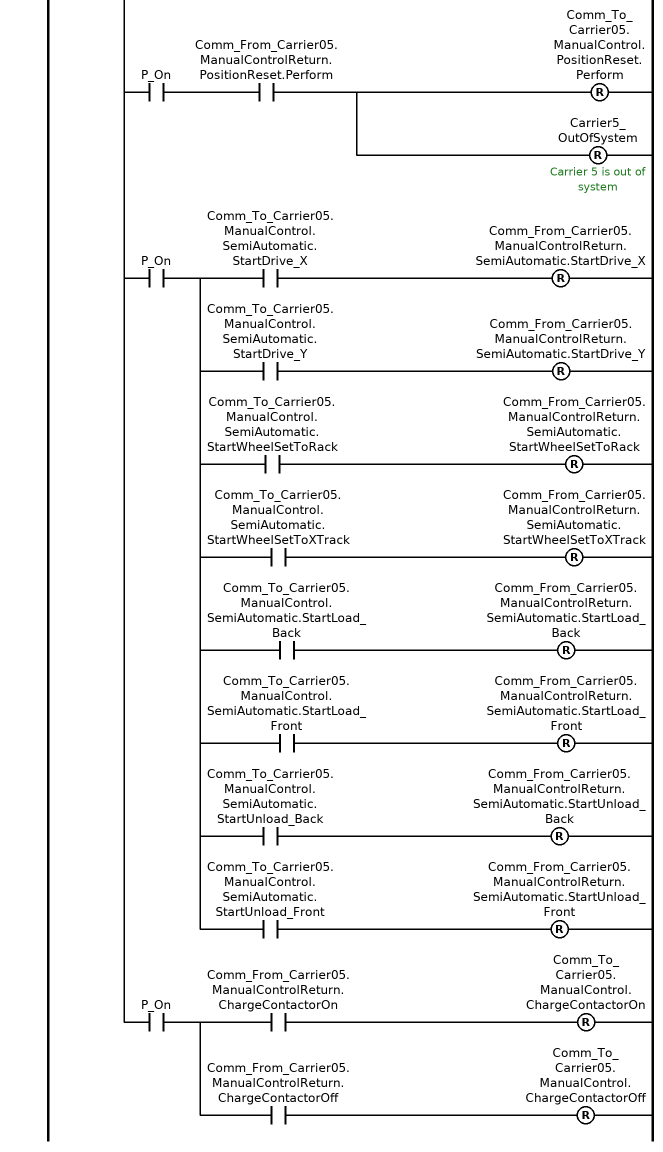
(* [picture p78: Mobile_Machines / Carrier05, rungs 8-8] *)
(* Rung 8: Reset several bits that are set by Dat-A-Control but not reset *)
IF P_On AND P_On AND Comm_From_Carrier05.Various.ResetAlarm_Return THEN
    Comm_To_Carrier05.Dat_A_Control.Settings_In0.ResetAlarm := FALSE;
END_IF;
IF P_On AND P_On AND Comm_From_Carrier05.Various.ResetCycle_Return THEN
    Comm_To_Carrier05.Dat_A_Control.Settings_In0.ResetCycle := FALSE;
END_IF;
IF P_On AND P_On AND Comm_From_Carrier05.Various.AbortCharge_Return THEN
    Comm_To_Carrier05.Various.AbortCharge := FALSE;
END_IF;
IF P_On AND P_On AND ES_OK AND Comm_From_Carrier05.Various.ResetMachineOn THEN
    Comm_To_Carrier05.Dat_A_Control.Settings_In0.MachineOn := FALSE;
END_IF;
IF P_On AND P_On AND Comm_From_Carrier05.ManualControlReturn.DriveRack.Out THEN
    Comm_To_Carrier05.ManualControl.DriveRack.Out := FALSE;
END_IF;
IF P_On AND P_On AND Comm_From_Carrier05.ManualControlReturn.DriveRack.In THEN
    Comm_To_Carrier05.ManualControl.DriveRack.In := FALSE;
END_IF;
IF P_On AND P_On AND Comm_From_Carrier05.ManualControlReturn.DriveRack.Stop THEN
    Comm_To_Carrier05.ManualControl.DriveRack.Stop := FALSE;
END_IF;
IF P_On AND P_On AND Comm_From_Carrier05.ManualControlReturn.DriveRack_FindXTrack.Out THEN
    Comm_To_Carrier05.ManualControl.DriveRack_FindXTrack.Out := FALSE;
END_IF;
IF P_On AND P_On AND Comm_From_Carrier05.ManualControlReturn.DriveRack_FindXTrack.In THEN
    Comm_To_Carrier05.ManualControl.DriveRack_FindXTrack.In := FALSE;
END_IF;
IF P_On AND P_On AND Comm_From_Carrier05.ManualControlReturn.DriveRack_FindXTrack.Stop THEN
    Comm_To_Carrier05.ManualControl.DriveRack_FindXTrack.Stop := FALSE;
END_IF;
IF P_On AND P_On AND Comm_From_Carrier05.ManualControlReturn.DriveXtrack.Out THEN
    Comm_To_Carrier05.ManualControl.DriveXtrack.Out := FALSE;
END_IF;
IF P_On AND P_On AND Comm_From_Carrier05.ManualControlReturn.DriveXtrack.In THEN
    Comm_To_Carrier05.ManualControl.DriveXtrack.In := FALSE;
END_IF;
IF P_On AND P_On AND Comm_From_Carrier05.ManualControlReturn.DriveXtrack.Stop THEN
    Comm_To_Carrier05.ManualControl.DriveXtrack.Stop := FALSE;
END_IF;
IF P_On AND P_On AND Comm_From_Carrier05.ManualControlReturn.DriveXTrack_FindPosition.Out THEN
    Comm_To_Carrier05.ManualControl.DriveXTrack_FindPosition.Out := FALSE;
END_IF;
IF P_On AND P_On AND Comm_From_Carrier05.ManualControlReturn.DriveXTrack_FindPosition.In THEN
    Comm_To_Carrier05.ManualControl.DriveXTrack_FindPosition.In := FALSE;
END_IF;
IF P_On AND P_On AND Comm_From_Carrier05.ManualControlReturn.DriveXTrack_FindPosition.Stop THEN
    Comm_To_Carrier05.ManualControl.DriveXTrack_FindPosition.Stop := FALSE;
END_IF;
IF P_On AND P_On AND Comm_From_Carrier05.ManualControlReturn.Wheelset.Out THEN
    Comm_To_Carrier05.ManualControl.Wheelset.Out := FALSE;
END_IF;
IF P_On AND P_On AND Comm_From_Carrier05.ManualControlReturn.Wheelset.In THEN
    Comm_To_Carrier05.ManualControl.Wheelset.In := FALSE;
END_IF;
IF P_On AND P_On AND Comm_From_Carrier05.ManualControlReturn.Wheelset.Stop THEN
    Comm_To_Carrier05.ManualControl.Wheelset.Stop := FALSE;
END_IF;
IF P_On AND P_On AND Comm_From_Carrier05.ManualControlReturn.LIftingPlate.UpMIN THEN
    Comm_To_Carrier05.ManualControl.LIftingPlate.UpMIN := FALSE;
END_IF;
IF P_On AND P_On AND Comm_From_Carrier05.ManualControlReturn.LIftingPlate.DownMIN THEN
    Comm_To_Carrier05.ManualControl.LIftingPlate.DownMIN := FALSE;
END_IF;
IF P_On AND P_On AND Comm_From_Carrier05.ManualControlReturn.LIftingPlate.StopMIN THEN
    Comm_To_Carrier05.ManualControl.LIftingPlate.StopMIN := FALSE;
END_IF;
IF P_On AND P_On AND Comm_From_Carrier05.ManualControlReturn.LIftingPlate.UpMAX THEN
    Comm_To_Carrier05.ManualControl.LIftingPlate.UpMAX := FALSE;
END_IF;
IF P_On AND P_On AND Comm_From_Carrier05.ManualControlReturn.LIftingPlate.DownMAX THEN
    Comm_To_Carrier05.ManualControl.LIftingPlate.DownMAX := FALSE;
END_IF;
IF P_On AND P_On AND Comm_From_Carrier05.ManualControlReturn.LIftingPlate.StopMAX THEN
    Comm_To_Carrier05.ManualControl.LIftingPlate.StopMAX := FALSE;
END_IF;
IF P_On AND P_On AND Comm_From_Carrier05.ManualControlReturn.LIftingPlate.UpBoth THEN
    Comm_To_Carrier05.ManualControl.LIftingPlate.UpBoth := FALSE;
END_IF;
IF P_On AND P_On AND Comm_From_Carrier05.ManualControlReturn.LIftingPlate.DownBoth THEN
    Comm_To_Carrier05.ManualControl.LIftingPlate.DownBoth := FALSE;
END_IF;
IF P_On AND P_On AND Comm_From_Carrier05.ManualControlReturn.LIftingPlate.StopBoth THEN
    Comm_To_Carrier05.ManualControl.LIftingPlate.StopBoth := FALSE;
END_IF;
_p59 := P_On AND P_On AND Comm_From_Carrier05.ManualControlReturn.PositionReset.Perform;
IF _p59 THEN
    Comm_To_Carrier05.ManualControl.PositionReset.Perform := FALSE;
    Carrier5_OutOfSystem := FALSE;
END_IF;
IF P_On AND P_On AND Comm_To_Carrier05.ManualControl.SemiAutomatic.StartDrive_X THEN
    Comm_From_Carrier05.ManualControlReturn.SemiAutomatic.StartDrive_X := FALSE;
END_IF;
IF P_On AND P_On AND Comm_To_Carrier05.ManualControl.SemiAutomatic.StartDrive_Y THEN
    Comm_From_Carrier05.ManualControlReturn.SemiAutomatic.StartDrive_Y := FALSE;
END_IF;
IF P_On AND P_On AND Comm_To_Carrier05.ManualControl.SemiAutomatic.StartWheelSetToRack THEN
    Comm_From_Carrier05.ManualControlReturn.SemiAutomatic.StartWheelSetToRack := FALSE;
END_IF;
IF P_On AND P_On AND Comm_To_Carrier05.ManualControl.SemiAutomatic.StartWheelSetToXTrack THEN
    Comm_From_Carrier05.ManualControlReturn.SemiAutomatic.StartWheelSetToXTrack := FALSE;
END_IF;
IF P_On AND P_On AND Comm_To_Carrier05.ManualControl.SemiAutomatic.StartLoad_Back THEN
    Comm_From_Carrier05.ManualControlReturn.SemiAutomatic.StartLoad_Back := FALSE;
END_IF;
IF P_On AND P_On AND Comm_To_Carrier05.ManualControl.SemiAutomatic.StartLoad_Front THEN
    Comm_From_Carrier05.ManualControlReturn.SemiAutomatic.StartLoad_Front := FALSE;
END_IF;
IF P_On AND P_On AND Comm_To_Carrier05.ManualControl.SemiAutomatic.StartUnload_Back THEN
    Comm_From_Carrier05.ManualControlReturn.SemiAutomatic.StartUnload_Back := FALSE;
END_IF;
IF P_On AND P_On AND Comm_To_Carrier05.ManualControl.SemiAutomatic.StartUnload_Front THEN
    Comm_From_Carrier05.ManualControlReturn.SemiAutomatic.StartUnload_Front := FALSE;
END_IF;
IF P_On AND P_On AND Comm_From_Carrier05.ManualControlReturn.ChargeContactorOn THEN
    Comm_To_Carrier05.ManualControl.ChargeContactorOn := FALSE;
END_IF;
IF P_On AND P_On AND Comm_From_Carrier05.ManualControlReturn.ChargeContactorOff THEN
    Comm_To_Carrier05.ManualControl.ChargeContactorOff := FALSE;
END_IF;

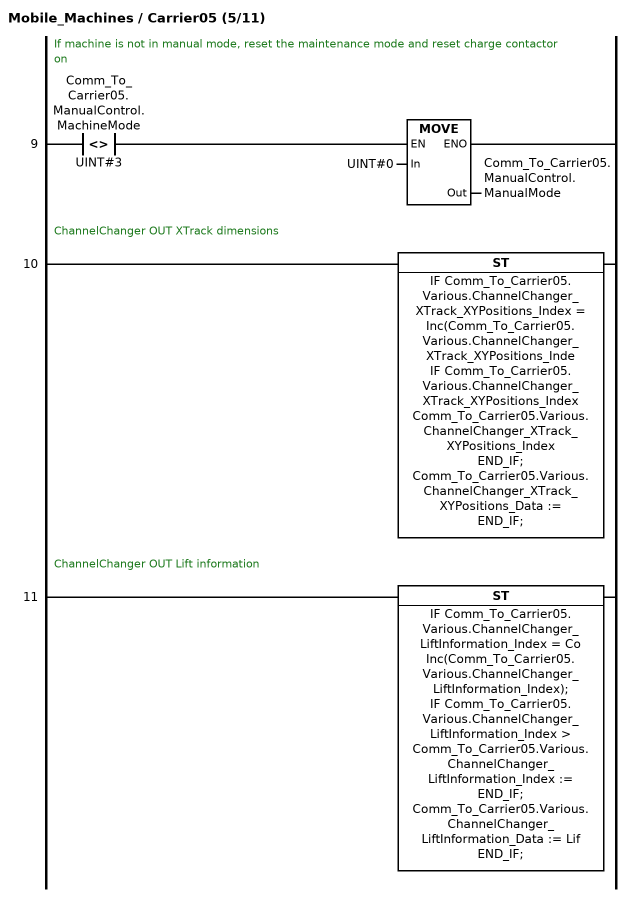
(* Rung 9: If machine is not in manual mode, reset the maintenance mode and reset charge contactor on *)
IF Comm_To_Carrier05.ManualControl.MachineMode <> UINT#3 THEN
    Comm_To_Carrier05.ManualControl.ManualMode := UINT#0;
END_IF;
(* Rung 10: ChannelChanger OUT XTrack dimensions *)
IF Comm_To_Carrier05.Various.ChannelChanger_XTrack_XYPositions_Index = Comm_From_Carrier05.Various.ChannelChanger_XTrack_XYPositions_Index THEN
	Inc(Comm_To_Carrier05.Various.ChannelChanger_XTrack_XYPositions_Index);
	IF Comm_To_Carrier05.Various.ChannelChanger_XTrack_XYPositions_Index > 199 THEN
		Comm_To_Carrier05.Various.ChannelChanger_XTrack_XYPositions_Index := 0;
	END_IF;
	Comm_To_Carrier05.Various.ChannelChanger_XTrack_XYPositions_Data := XTrack_XYPositions_Array[Comm_To_Carrier05.Various.ChannelChanger_XTrack_XYPositions_Index];
END_IF;
(* Rung 11: ChannelChanger OUT Lift information *)
IF Comm_To_Carrier05.Various.ChannelChanger_LiftInformation_Index = Comm_From_Carrier05.Various.ChannelChanger_LiftInformation_Index THEN
	Inc(Comm_To_Carrier05.Various.ChannelChanger_LiftInformation_Index);
	IF Comm_To_Carrier05.Various.ChannelChanger_LiftInformation_Index > 99 THEN
		Comm_To_Carrier05.Various.ChannelChanger_LiftInformation_Index := 0;
	END_IF;
	Comm_To_Carrier05.Various.ChannelChanger_LiftInformation_Data := Lift_Array[Comm_To_Carrier05.Various.ChannelChanger_LiftInformation_Index];
END_IF;

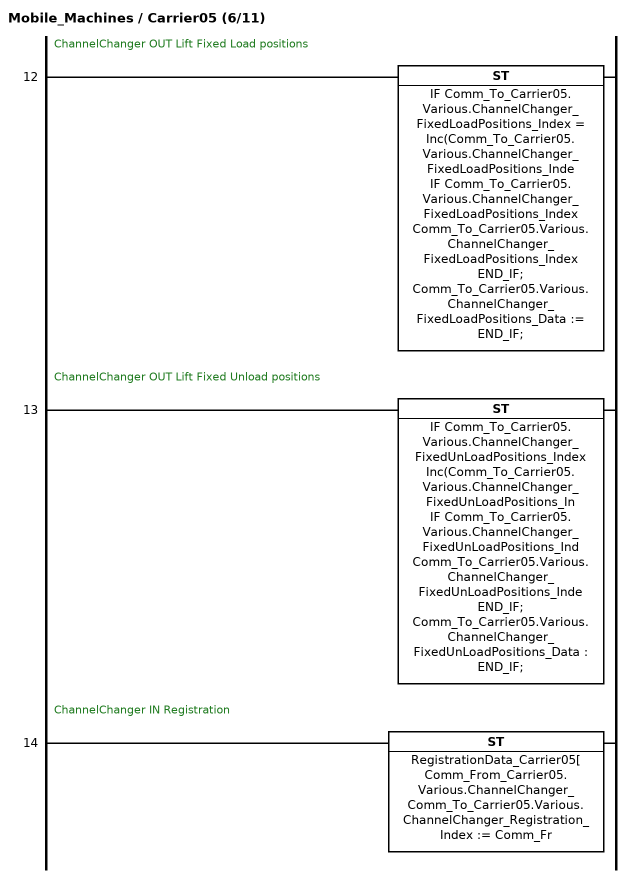
(* Rung 12: ChannelChanger OUT Lift Fixed Load positions *)
IF Comm_To_Carrier05.Various.ChannelChanger_FixedLoadPositions_Index = Comm_From_Carrier05.Various.ChannelChanger_FixedLoadPositions_Index THEN
	Inc(Comm_To_Carrier05.Various.ChannelChanger_FixedLoadPositions_Index);
	IF Comm_To_Carrier05.Various.ChannelChanger_FixedLoadPositions_Index > 199 THEN
		Comm_To_Carrier05.Various.ChannelChanger_FixedLoadPositions_Index := 0;
	END_IF;
	Comm_To_Carrier05.Various.ChannelChanger_FixedLoadPositions_Data := FixedLoadPosition_Array[Comm_To_Carrier05.Various.ChannelChanger_FixedLoadPositions_Index];
END_IF;
(* Rung 13: ChannelChanger OUT Lift Fixed Unload positions *)
IF Comm_To_Carrier05.Various.ChannelChanger_FixedUnLoadPositions_Index = Comm_From_Carrier05.Various.ChannelChanger_FixedUnLoadPositions_Index THEN
	Inc(Comm_To_Carrier05.Various.ChannelChanger_FixedUnLoadPositions_Index);
	IF Comm_To_Carrier05.Various.ChannelChanger_FixedUnLoadPositions_Index > 199 THEN
		Comm_To_Carrier05.Various.ChannelChanger_FixedUnLoadPositions_Index := 0;
	END_IF;
	Comm_To_Carrier05.Various.ChannelChanger_FixedUnLoadPositions_Data := FixedUnloadPosition_Array[Comm_To_Carrier05.Various.ChannelChanger_FixedUnLoadPositions_Index];
END_IF;
(* Rung 14: ChannelChanger IN Registration *)
RegistrationData_Carrier05[Comm_From_Carrier05.Various.ChannelChanger_Registration_Index] := Comm_From_Carrier05.Various.ChannelChanger_Registration_Data;
Comm_To_Carrier05.Various.ChannelChanger_Registration_Index := Comm_From_Carrier05.Various.ChannelChanger_Registration_Index;

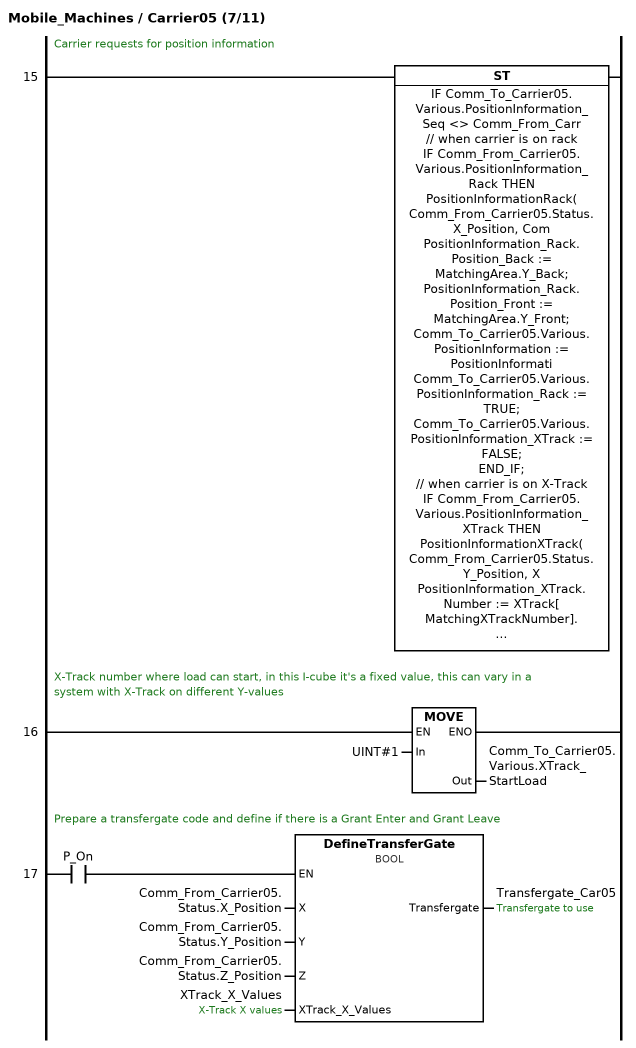
(* Rung 15: Carrier requests for position information *)
IF Comm_To_Carrier05.Various.PositionInformation_Seq <> Comm_From_Carrier05.Various.PositionInformation_Seq THEN
	// when carrier is on rack
	IF Comm_From_Carrier05.Various.PositionInformation_Rack THEN
		PositionInformationRack(Comm_From_Carrier05.Status.X_Position, Comm_From_Carrier05.Status.Y_Position, Comm_From_Carrier05.Status.Z_Position, Settings_CP.Margin_AreaCompare, Area, MatchingArea);
		PositionInformation_Rack.Position_Back := MatchingArea.Y_Back;
		PositionInformation_Rack.Position_Front := MatchingArea.Y_Front;
		Comm_To_Carrier05.Various.PositionInformation := PositionInformation_Rough;
		Comm_To_Carrier05.Various.PositionInformation_Rack := TRUE;
		Comm_To_Carrier05.Various.PositionInformation_XTrack := FALSE;
	END_IF;
	
	// when carrier is on X-Track
	IF Comm_From_Carrier05.Various.PositionInformation_XTrack THEN
		PositionInformationXTrack(Comm_From_Carrier05.Status.Y_Position, XTrack_Y_Values, MatchingXTrackNumber);
		PositionInformation_XTrack.Number := XTrack[MatchingXTrackNumber].XTrack_Number;
		PositionInformation_XTrack.Position_MIN := XTrack[MatchingXTrackNumber].MinimumPosition;
		PositionInformation_XTrack.Position_MAX := XTrack[MatchingXTrackNumber].MaximumPosition;
		Comm_To_Carrier05.Various.PositionInformation := PositionInformation_Rough;
		Comm_To_Carrier05.Various.PositionInformation_Rack := FALSE;
		Comm_To_Carrier05.Various.PositionInformation_XTrack := TRUE;
	END_IF;
	
	Comm_To_Carrier05.Various.PositionInformation_Seq := Comm_From_Carrier05.Various.PositionInformation_Seq;
	
END_IF;
(* Rung 16: X-Track number where load can start, in this I-cube it's a fixed value, this can vary in a system with X-Track on different Y-values *)
Comm_To_Carrier05.Various.XTrack_StartLoad := UINT#1;
(* Rung 17: Prepare a transfergate code and define if there is a Grant Enter and Grant Leave *)
_t60 := FALSE;
IF P_On THEN _t60 := DefineTransferGate(X := Comm_From_Carrier05.Status.X_Position, Y := Comm_From_Carrier05.Status.Y_Position, Z := Comm_From_Carrier05.Status.Z_Position, XTrack_X_Values := XTrack_X_Values, Transfergate => Transfergate_Car05); END_IF;

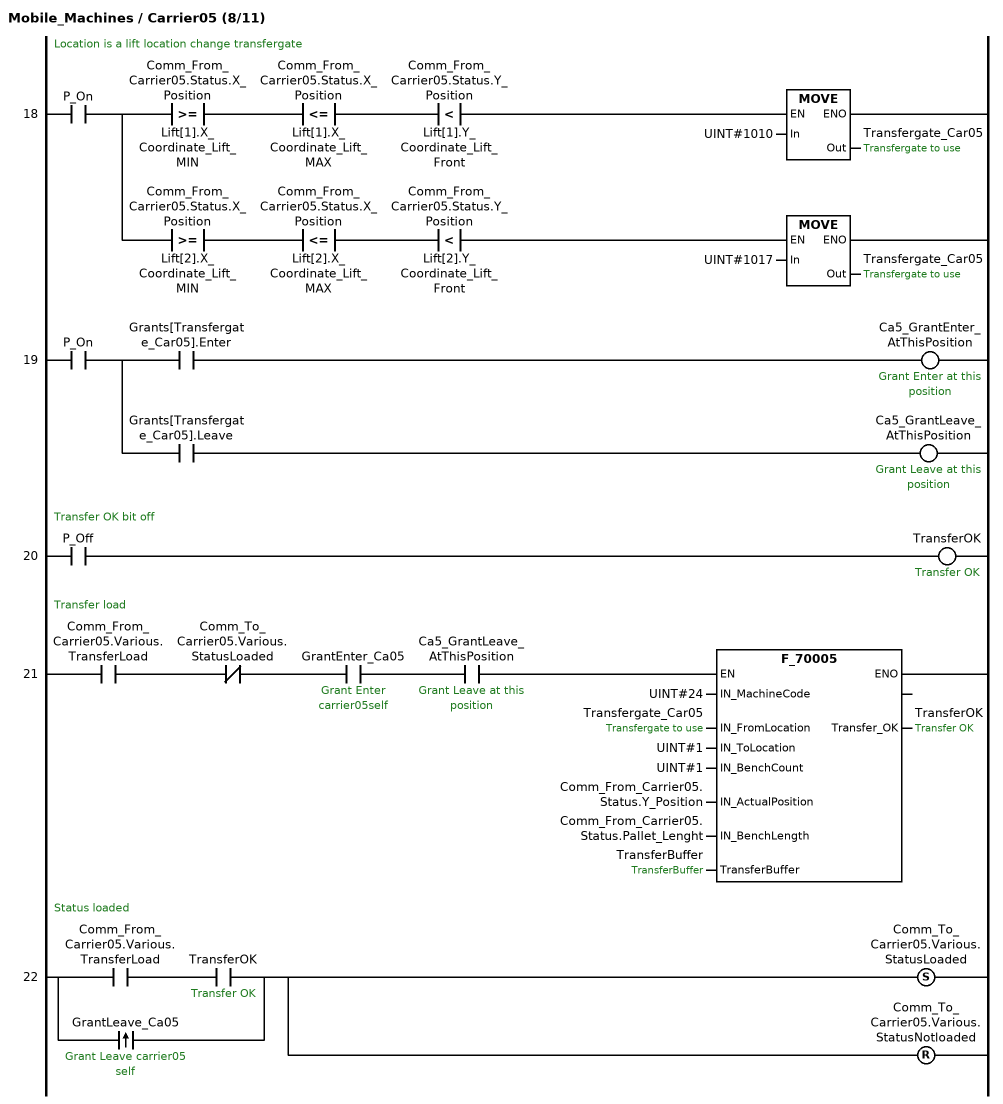
(* Rung 18: Location is a lift location change transfergate *)
IF P_On AND (Comm_From_Carrier05.Status.X_Position >= Lift[1].X_Coordinate_Lift_MIN) AND (Comm_From_Carrier05.Status.X_Position <= Lift[1].X_Coordinate_Lift_MAX) AND (Comm_From_Carrier05.Status.Y_Position < Lift[1].Y_Coordinate_Lift_Front) THEN
    Transfergate_Car05 := UINT#1010;
END_IF;
IF P_On AND (Comm_From_Carrier05.Status.X_Position >= Lift[2].X_Coordinate_Lift_MIN) AND (Comm_From_Carrier05.Status.X_Position <= Lift[2].X_Coordinate_Lift_MAX) AND (Comm_From_Carrier05.Status.Y_Position < Lift[2].Y_Coordinate_Lift_Front) THEN
    Transfergate_Car05 := UINT#1017;
END_IF;
(* Rung 19 *)
Ca5_GrantEnter_AtThisPosition := P_On AND Grants[Transfergate_Car05].Enter;
Ca5_GrantLeave_AtThisPosition := P_On AND Grants[Transfergate_Car05].Leave;
(* Rung 20: Transfer OK bit off *)
TransferOK := P_Off;
(* Rung 21: Transfer load *)
IF Comm_From_Carrier05.Various.TransferLoad AND NOT Comm_To_Carrier05.Various.StatusLoaded AND GrantEnter_Ca05 AND Ca5_GrantLeave_AtThisPosition THEN
    F_70005(IN_MachineCode := UINT#24, IN_FromLocation := Transfergate_Car05, IN_ToLocation := UINT#1, IN_BenchCount := UINT#1, IN_ActualPosition := Comm_From_Carrier05.Status.Y_Position, IN_BenchLength := Comm_From_Carrier05.Status.Pallet_Lenght, TransferBuffer := TransferBuffer, Transfer_OK => TransferOK);
END_IF;
(* Rung 22: Status loaded *)
_e61(CLK := GrantLeave_Ca05);
_p62 := (Comm_From_Carrier05.Various.TransferLoad AND TransferOK) OR _e61.Q;
IF _p62 THEN
    Comm_To_Carrier05.Various.StatusLoaded := TRUE;
    Comm_To_Carrier05.Various.StatusNotloaded := FALSE;
END_IF;

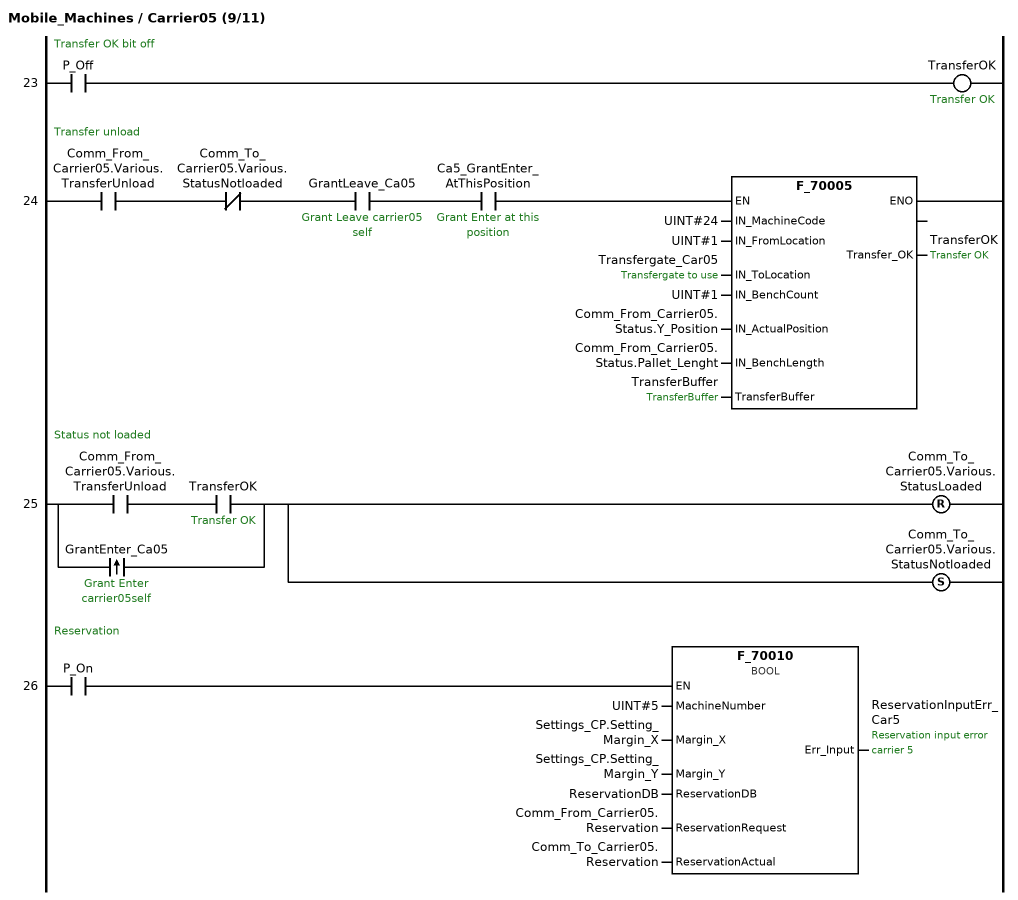
(* Rung 23: Transfer OK bit off *)
TransferOK := P_Off;
(* Rung 24: Transfer unload *)
IF Comm_From_Carrier05.Various.TransferUnload AND NOT Comm_To_Carrier05.Various.StatusNotloaded AND GrantLeave_Ca05 AND Ca5_GrantEnter_AtThisPosition THEN
    F_70005(IN_MachineCode := UINT#24, IN_FromLocation := UINT#1, IN_ToLocation := Transfergate_Car05, IN_BenchCount := UINT#1, IN_ActualPosition := Comm_From_Carrier05.Status.Y_Position, IN_BenchLength := Comm_From_Carrier05.Status.Pallet_Lenght, TransferBuffer := TransferBuffer, Transfer_OK => TransferOK);
END_IF;
(* Rung 25: Status not loaded *)
_e63(CLK := GrantEnter_Ca05);
_p64 := (Comm_From_Carrier05.Various.TransferUnload AND TransferOK) OR _e63.Q;
IF _p64 THEN
    Comm_To_Carrier05.Various.StatusLoaded := FALSE;
    Comm_To_Carrier05.Various.StatusNotloaded := TRUE;
END_IF;
(* Rung 26: Reservation *)
_t65 := FALSE;
IF P_On THEN _t65 := F_70010(MachineNumber := UINT#5, Margin_X := Settings_CP.Setting_Margin_X, Margin_Y := Settings_CP.Setting_Margin_Y, ReservationDB := ReservationDB, ReservationRequest := Comm_From_Carrier05.Reservation, ReservationActual := Comm_To_Carrier05.Reservation, Err_Input => ReservationInputErr_Car5); END_IF;

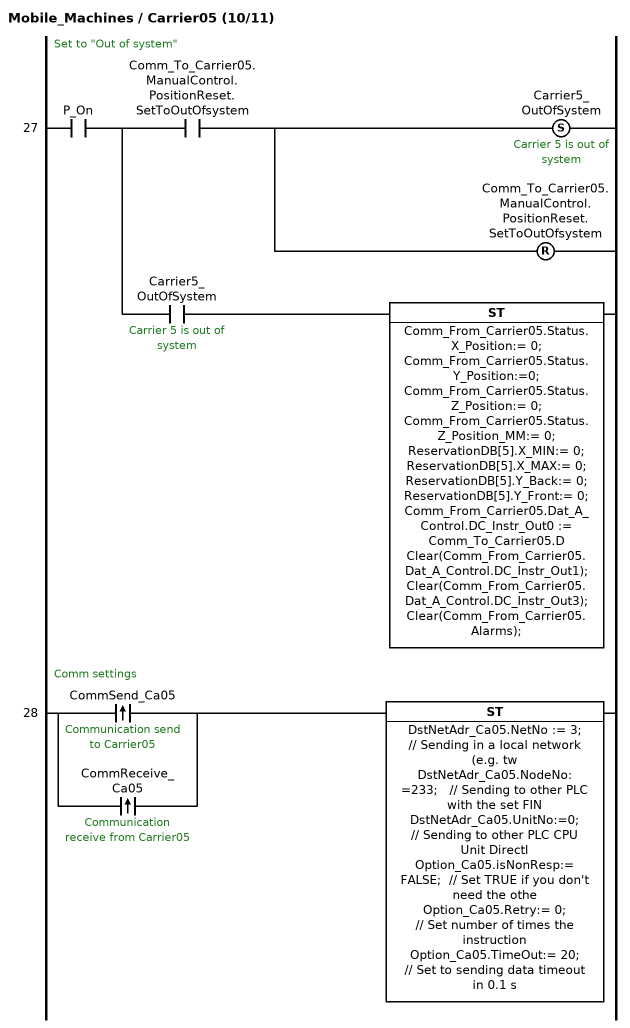
(* Rung 27: Set to "Out of system" *)
_p66 := P_On AND Comm_To_Carrier05.ManualControl.PositionReset.SetToOutOfsystem;
IF _p66 THEN
    Carrier5_OutOfSystem := TRUE;
    Comm_To_Carrier05.ManualControl.PositionReset.SetToOutOfsystem := FALSE;
END_IF;
IF P_On AND Carrier5_OutOfSystem THEN
    Comm_From_Carrier05.Status.X_Position:= 0;
    Comm_From_Carrier05.Status.Y_Position:=0;
    Comm_From_Carrier05.Status.Z_Position:= 0;
    Comm_From_Carrier05.Status.Z_Position_MM:= 0;
    
    ReservationDB[5].X_MIN:= 0;
    ReservationDB[5].X_MAX:= 0;
    ReservationDB[5].Y_Back:= 0;
    ReservationDB[5].Y_Front:= 0;
    
    Comm_From_Carrier05.Dat_A_Control.DC_Instr_Out0 := Comm_To_Carrier05.Dat_A_Control.Instr_Sequencenumber;
    Clear(Comm_From_Carrier05.Dat_A_Control.DC_Instr_Out1);
    Clear(Comm_From_Carrier05.Dat_A_Control.DC_Instr_Out3);
    Clear(Comm_From_Carrier05.Alarms);
END_IF;
(* Rung 28: Comm settings *)
_e67(CLK := CommSend_Ca05);
_e68(CLK := CommReceive_Ca05);
IF _e67.Q OR _e68.Q THEN
    DstNetAdr_Ca05.NetNo := 3;			// Sending in a local network (e.g. two PLCs connected by Ethernet LAN vai a hub)
    DstNetAdr_Ca05.NodeNo:=233;		// Sending to other PLC with the set FINS Node NUmber (depending on the other PLC)
    DstNetAdr_Ca05.UnitNo:=0;			// Sending to other PLC CPU Unit Directly
    
    Option_Ca05.isNonResp:= FALSE; 	// Set TRUE if you don't need the other CPU to reply back, otherwise set to FALSE
    Option_Ca05.Retry:= 0;					// Set number of times the instruction will retry sending if it failed to send data
    Option_Ca05.TimeOut:= 20;			// Set to sending data timeout in 0.1 s unit (e.g. 20 = 2 secs)
END_IF;

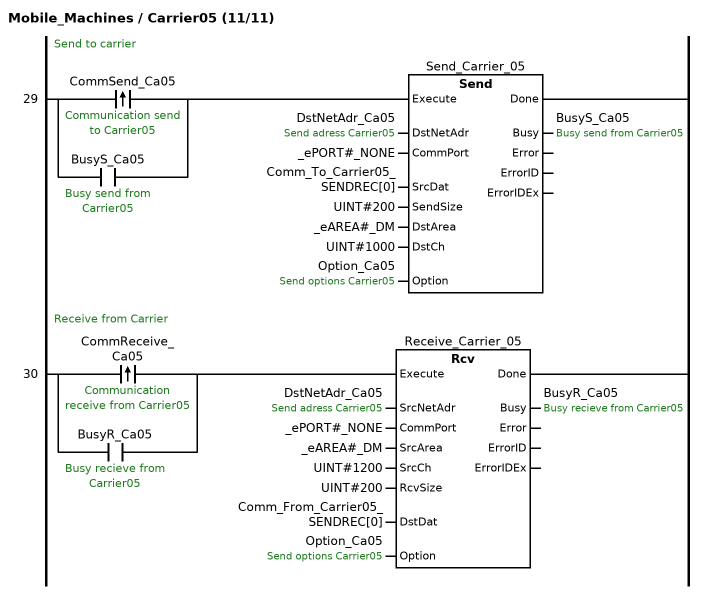
(* Rung 29: Send to carrier *)
_e69(CLK := CommSend_Ca05);
Send_Carrier_05(Execute := _e69.Q OR BusyS_Ca05, DstNetAdr := DstNetAdr_Ca05, CommPort := _ePORT#_NONE, SrcDat := Comm_To_Carrier05_SENDREC[0], SendSize := UINT#200, DstArea := _eAREA#_DM, DstCh := UINT#1000, Option := Option_Ca05, Busy => BusyS_Ca05);
(* Rung 30: Receive from Carrier *)
_e70(CLK := CommReceive_Ca05);
Receive_Carrier_05(Execute := _e70.Q OR BusyR_Ca05, SrcNetAdr := DstNetAdr_Ca05, CommPort := _ePORT#_NONE, SrcArea := _eAREA#_DM, SrcCh := UINT#1200, RcvSize := UINT#200, DstDat := Comm_From_Carrier05_SENDREC[0], Option := Option_Ca05, Busy => BusyR_Ca05);

(* Section Chargers: ladder, written here as Structured Text *)

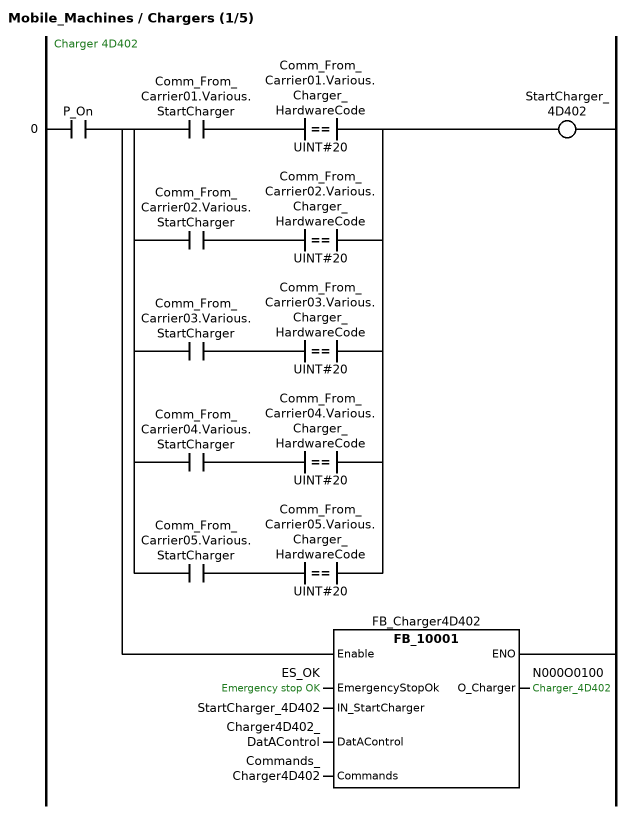
(* Rung 0: Charger 4D402 *)
StartCharger_4D402 := P_On AND ((Comm_From_Carrier01.Various.StartCharger AND (Comm_From_Carrier01.Various.Charger_HardwareCode = UINT#20)) OR (Comm_From_Carrier02.Various.StartCharger AND (Comm_From_Carrier02.Various.Charger_HardwareCode = UINT#20)) OR (Comm_From_Carrier03.Various.StartCharger AND (Comm_From_Carrier03.Various.Charger_HardwareCode = UINT#20)) OR (Comm_From_Carrier04.Various.StartCharger AND (Comm_From_Carrier04.Various.Charger_HardwareCode = UINT#20)) OR (Comm_From_Carrier05.Various.StartCharger AND (Comm_From_Carrier05.Various.Charger_HardwareCode = UINT#20)));
FB_Charger4D402(Enable := P_On, EmergencyStopOk := ES_OK, IN_StartCharger := StartCharger_4D402, DatAControl := Charger4D402_DatAControl, Commands := Commands_Charger4D402, O_Charger => N000O0100);

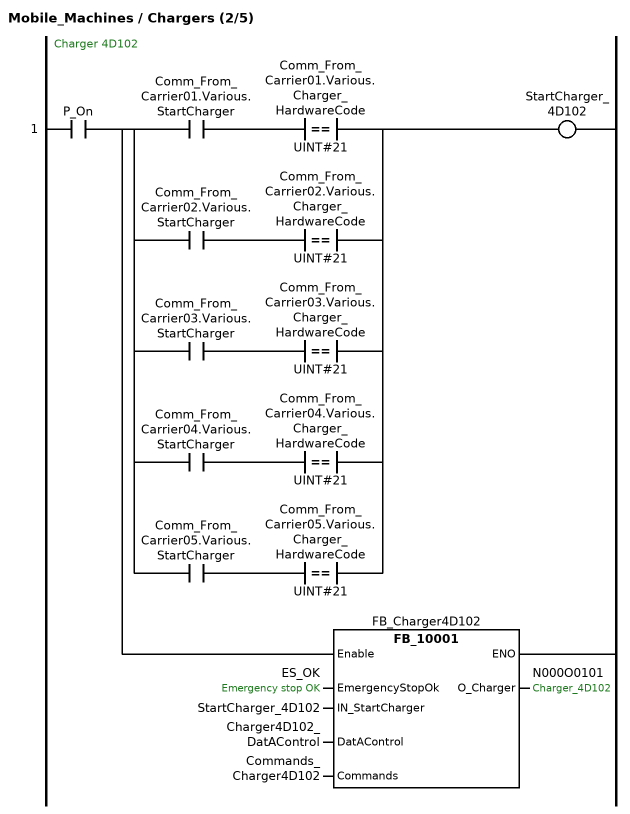
(* Rung 1: Charger 4D102 *)
StartCharger_4D102 := P_On AND ((Comm_From_Carrier01.Various.StartCharger AND (Comm_From_Carrier01.Various.Charger_HardwareCode = UINT#21)) OR (Comm_From_Carrier02.Various.StartCharger AND (Comm_From_Carrier02.Various.Charger_HardwareCode = UINT#21)) OR (Comm_From_Carrier03.Various.StartCharger AND (Comm_From_Carrier03.Various.Charger_HardwareCode = UINT#21)) OR (Comm_From_Carrier04.Various.StartCharger AND (Comm_From_Carrier04.Various.Charger_HardwareCode = UINT#21)) OR (Comm_From_Carrier05.Various.StartCharger AND (Comm_From_Carrier05.Various.Charger_HardwareCode = UINT#21)));
FB_Charger4D102(Enable := P_On, EmergencyStopOk := ES_OK, IN_StartCharger := StartCharger_4D102, DatAControl := Charger4D102_DatAControl, Commands := Commands_Charger4D102, O_Charger => N000O0101);

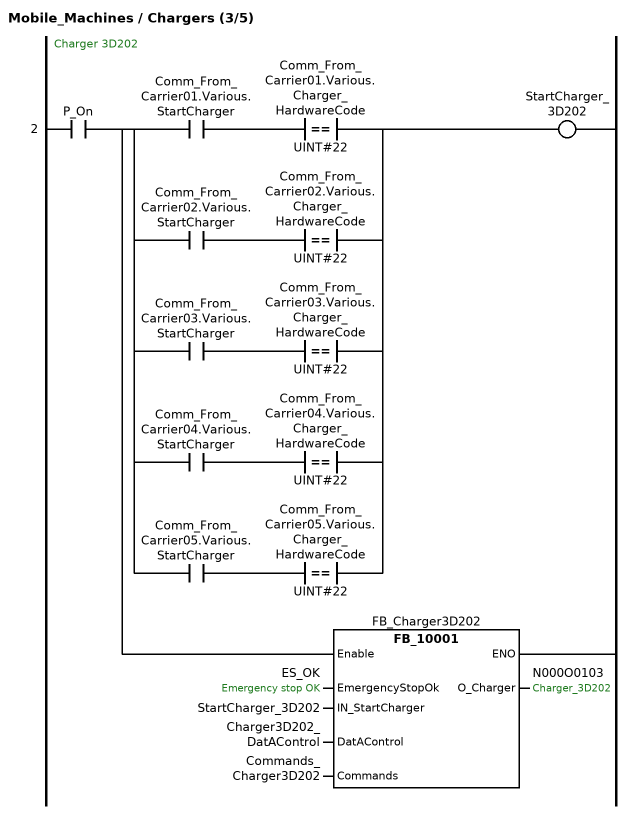
(* Rung 2: Charger 3D202 *)
StartCharger_3D202 := P_On AND ((Comm_From_Carrier01.Various.StartCharger AND (Comm_From_Carrier01.Various.Charger_HardwareCode = UINT#22)) OR (Comm_From_Carrier02.Various.StartCharger AND (Comm_From_Carrier02.Various.Charger_HardwareCode = UINT#22)) OR (Comm_From_Carrier03.Various.StartCharger AND (Comm_From_Carrier03.Various.Charger_HardwareCode = UINT#22)) OR (Comm_From_Carrier04.Various.StartCharger AND (Comm_From_Carrier04.Various.Charger_HardwareCode = UINT#22)) OR (Comm_From_Carrier05.Various.StartCharger AND (Comm_From_Carrier05.Various.Charger_HardwareCode = UINT#22)));
FB_Charger3D202(Enable := P_On, EmergencyStopOk := ES_OK, IN_StartCharger := StartCharger_3D202, DatAControl := Charger3D202_DatAControl, Commands := Commands_Charger3D202, O_Charger => N000O0103);

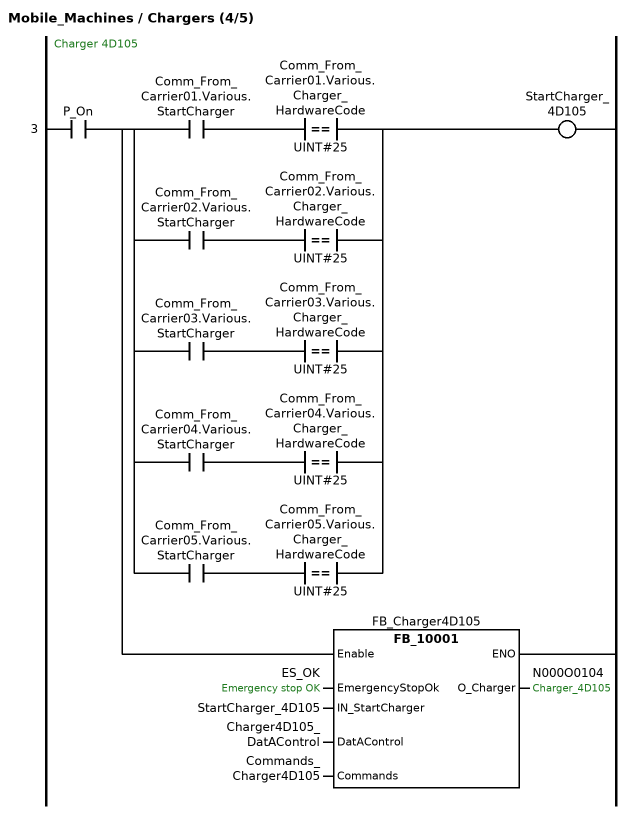
(* Rung 3: Charger 4D105 *)
StartCharger_4D105 := P_On AND ((Comm_From_Carrier01.Various.StartCharger AND (Comm_From_Carrier01.Various.Charger_HardwareCode = UINT#25)) OR (Comm_From_Carrier02.Various.StartCharger AND (Comm_From_Carrier02.Various.Charger_HardwareCode = UINT#25)) OR (Comm_From_Carrier03.Various.StartCharger AND (Comm_From_Carrier03.Various.Charger_HardwareCode = UINT#25)) OR (Comm_From_Carrier04.Various.StartCharger AND (Comm_From_Carrier04.Various.Charger_HardwareCode = UINT#25)) OR (Comm_From_Carrier05.Various.StartCharger AND (Comm_From_Carrier05.Various.Charger_HardwareCode = UINT#25)));
FB_Charger4D105(Enable := P_On, EmergencyStopOk := ES_OK, IN_StartCharger := StartCharger_4D105, DatAControl := Charger4D105_DatAControl, Commands := Commands_Charger4D105, O_Charger => N000O0104);

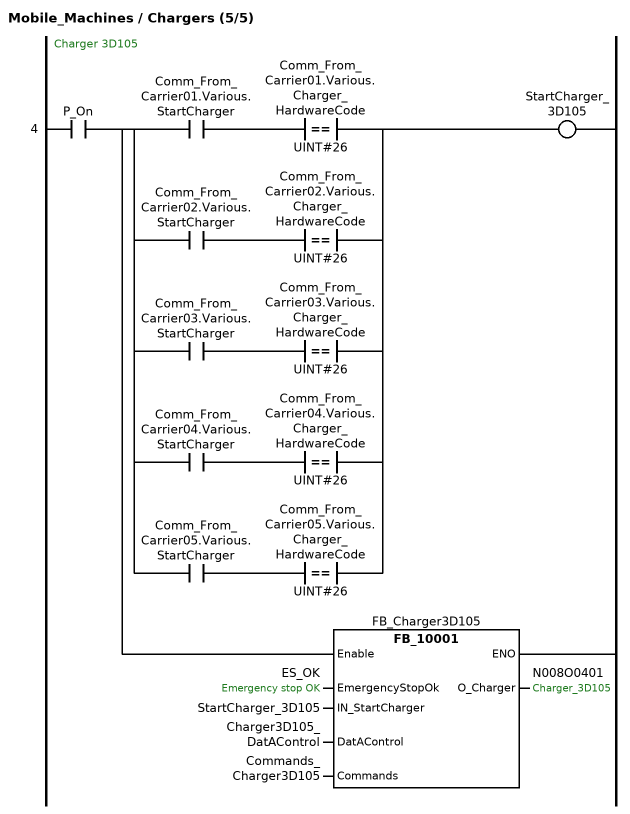
(* Rung 4: Charger 3D105 *)
StartCharger_3D105 := P_On AND ((Comm_From_Carrier01.Various.StartCharger AND (Comm_From_Carrier01.Various.Charger_HardwareCode = UINT#26)) OR (Comm_From_Carrier02.Various.StartCharger AND (Comm_From_Carrier02.Various.Charger_HardwareCode = UINT#26)) OR (Comm_From_Carrier03.Various.StartCharger AND (Comm_From_Carrier03.Various.Charger_HardwareCode = UINT#26)) OR (Comm_From_Carrier04.Various.StartCharger AND (Comm_From_Carrier04.Various.Charger_HardwareCode = UINT#26)) OR (Comm_From_Carrier05.Various.StartCharger AND (Comm_From_Carrier05.Various.Charger_HardwareCode = UINT#26)));
FB_Charger3D105(Enable := P_On, EmergencyStopOk := ES_OK, IN_StartCharger := StartCharger_3D105, DatAControl := Charger3D105_DatAControl, Commands := Commands_Charger3D105, O_Charger => N008O0401);
END_PROGRAM

PROGRAM Work_Level01
VAR
    Belt_W02 : FB_25050;
    SettingsW02 : ST_FB_25050\Settings;  (* Settings W02 *)
    W02_WriteParameter : BOOL;  (* Write inverter parameters *)
    W02_WriteParametersDone : BOOL;  (* Write inverter parameters is done *)
    T01W02_InverterParameters : ST_MX2\Parameters;  (* Inverter parameters *)
    T01W02_WriteParameters : BOOL;  (* Write parameters *)
    T01W02_WriteParametersDone : BOOL;  (* Write parameters done *)
    SettingsW01 : ST_FB_25050\Settings;  (* Settings W01 *)
    Belt_W01 : FB_25050;
    W01_WriteParameters : BOOL;
    W01_WriteParameterDone : BOOL;
    T01W01 : FB_30052;
    T01W01_Inputs : ST_FB_30050_Inputs;  (* Inputs T01W01 *)
    T01W02_Inputs : ST_FB_30050_Inputs;  (* Inputs T01W02 *)
    T01W02_Settings : ST_FB_30052_Settings;  (* Settings T01W02 *)
    T01W01_WriteParameters : BOOL;  (* Write parameters *)
    T01W01_WriteParametersDone : BOOL;  (* Write parameters done *)
    Comm_From_W01 : ST_FB_30051_CommInPipe;  (* Comm from W01 *)
    Comm_To_W01 : ST_FB_30051_CommOutPipe;  (* Comm to W01 *)
    Comm_From_W02 : ST_FB_30051_CommInPipe;  (* Comm from W02 *)
    Comm_To_W02 : ST_FB_30051_CommOutPipe;  (* Comm to W02 *)
    T01W01_Settings : ST_FB_30052_Settings;  (* Settings T01W01 *)
    T01W02 : FB_30052;
    CommOut_T01W01_202 : ST_FB_30051_CommOut202;  (* Comm out 202 *)
    CommOut_T01W02_201 : ST_FB_30051_CommOut201;
    T01W01iTrack_201 : FB_101;
    T01W01iTrack201DON : BOOL;  (* Sensor track 201 time delay on *)
    T01W01iTrack201DOFF : BOOL;  (* Sensor track 201 time delay off *)
    T01W01iTrack_202 : FB_101;
    T01W01iTrack202DON : BOOL;  (* Sensor track 202 time delay on *)
    T01W01iTrack202DOFF : BOOL;  (* Sensor track 202 time delay off *)
    T01W02iTrack_201 : FB_101;
    T01W02iTrack201DON : BOOL;  (* Sensor track 201 time delay on *)
    T01W02iTrack201DOFF : BOOL;  (* Sensor track 201 time delay off *)
    T01W02iTrack_202 : FB_101;
    T01W02iTrack202DON : BOOL;  (* Sensor track 202 time delay on *)
    T01W02iTrack202DOFF : BOOL;  (* Sensor track 202 time delay off *)
    OutputsT01W01 : ST_FB_30052_Outputs;
    OutputsT01W02 : ST_FB_30052_Outputs;
    test_me : BOOL;
    test_me1 : BOOL;
END_VAR
VAR_EXTERNAL
    Dummy : BOOL;
    ES_OK : BOOL;
    W02_Dat_A_Control : ST_DatAControl_Standard;  (* Dat-A-Control interface *)
    W02_Commands : ST_FB_25050\Commands;  (* Commands W02 *)
    InverterStatus_Belt_W02 : ST_MX2\Status;  (* Inverter ststus *)
    InverterInputs_Belt_W02 : ST_MX2\Input;
    InverterCommands_Belt_W02 : ST_MX2\Command;  (* Commnads inverter Belt W02 *)
    InverterSpeed_Belt_W02 : INT;  (* Inverter speed belt W02 *)
    Comm_T01W02_W02 : ST_FB_25050\CommInPipe;  (* Communication from T01W02 to W02 *)
    Comm_LiftGR4_W02 : ST_FB_25050\CommInPipe;  (* Communication from liftGR4 to W02 *)
    Comm_W02_T01W02 : ST_FB_25050\CommOutPipe;  (* Communication from W02 to T01W02 *)
    Comm_W02_LiftGR04 : ST_FB_25050\CommOutPipe;  (* Communication from W02 to LiftGR4 *)
    T01W02_Dat_A_Control : ST_DatAControl_Standard;  (* IN.MachineMode Machine mode; IN.Settings.ResetAlarm Reset Alarm; OUT.TotalDone Total Done; OUT.Alarm00 Alarm word 0; OUT.Alarm01 Alarm word 1; IN.Instruction Instruction; IN Instruction; IN.Settings.ResetCycle Reset cycle; OUT.Alarm03 Alarm word 3; OUT.Alarm02 Alarmword 2 *)
    T01W02_Commands : ST_FB_30051_Commands;
    InverterStatus_T01W02 : ST_MX2\Status;  (* Inverter status *)
    InverterCommands_T01W02 : ST_MX2\Command;  (* Inverter commands *)
    InverterSpeed_T01W02 : INT;  (* Inverter speed *)
    T01W02_Direction : UINT;  (* Track direction 1 = to growroom 2 = To workarea *)
    InverterInputs_T01W02 : ST_MX2\Input;
    InverterOutputs_T01W02 : ST_MX2\Output;
    TransferBuffer : ST_TransferBuffer;
    InverterStatus_Belt_W01 : ST_MX2\Status;  (* Inverter status w01 *)
    InverterInputs_Belt_W01 : ST_MX2\Input;
    InverterCommands_Belt_W01 : ST_MX2\Command;  (* Commands inverter belt W01 *)
    InverterSpeed_Belt_W01 : INT;
    W01_Commands : ST_FB_25050\Commands;  (* Commands W01 *)
    W01_Dat_A_Control : ST_DatAControl_Standard;  (* Dat-A-Control interface *)
    Comm_LiftGR3_W01 : ST_FB_25050\CommInPipe;  (* Communication from liftGR3 to W01 *)
    Comm_T01W01_W01 : ST_FB_25050\CommInPipe;  (* Communication from T01W01 to W01 *)
    Comm_W01_LiftGR3 : ST_FB_25050\CommOutPipe;  (* Communication from W01 to LiftGR3 *)
    Comm_W01_T01W01 : ST_FB_25050\CommOutPipe;  (* Communication from W01 to T01W01 *)
    InverterStatus_T01W01 : ST_MX2\Status;  (* Inverter status *)
    InverterCommands_T01W01 : ST_MX2\Command;  (* Inverter commands *)
    InverterSpeed_T01W01 : INT;  (* Inverter speed *)
    InverterOutputs_T01W01 : ST_MX2\Output;  (* Inverter outputs *)
    T01W01_Dat_A_Control : ST_DatAControl_Standard;  (* Dat-A-Control *)
    InverterInputs_T01W01 : ST_MX2\Input;
    T01W01_Commands : ST_FB_30051_Commands;
    T01W01_Direction : UINT;
    N045I0103 : BOOL;
    N045I0104 : BOOL;
    N045I0105 : BOOL;
    N045I0110 : BOOL;
    N045I0111 : BOOL;
    N045I0101 : BOOL;
    N045I0102 : BOOL;
    N045I0113 : BOOL;
    N045I0114 : BOOL;
    N045I0106 : BOOL;
    N045I0107 : BOOL;
    N045I0108 : BOOL;
    N045I0109 : BOOL;
    InverterStatus_CLE_Spray : ST_MX2\Status;
    InverterStatus_CLE_Dirt : ST_MX2\Status;
    InverterStatus_CLE_Turn : ST_MX2\Status;
    N045O0200 : BOOL;
    N045O0205 : BOOL;
    N045O0201 : BOOL;
    N045O0206 : BOOL;
    N045O0202 : BOOL;
    N045O0203 : BOOL;
    N045O0204 : BOOL;
    InverterSpeed_CLE_Turn : INT;
    N045O0210 : BOOL;
    N045I0100 : BOOL;
    N045O0207 : BOOL;
    N045O0208 : BOOL;
    N045O0209 : BOOL;
    InverterCommands_CLE_Dirt : ST_MX2\Command;
    InverterCommands_CLE_Spray : ST_MX2\Command;
    InverterCommands_CLE_Turn : ST_MX2\Command;
    InverterSpeed_CLE_Dirt : INT;
    InverterSpeed_CLE_Spray : INT;
    Stacker_DatAControl : ST_DatAControl_Standard;  (* Dat A Control; IN.MachineMode Machine mode; IN.Settings.ResetAlarm Reset alarm; OUT.Alarm01 Alarm 1; OUT.Alarm03 Alarm 3; IN.ManualMode Manual override *)
    InverterInputs_W04 : ST_MX2\Input;
    Comm_From_Carrier01 : ST_FB_40701\Comm_OUT;
    InverterStatus_W04 : ST_MX2\Status;
    InverterCommands_W04 : ST_MX2\Command;
    InverterSpeed_W04 : INT;
    InverterOutputs_W04 : ST_MX2\Output;
    Comm_T01_T01W01 : ST_FB_30051_CommIn202;
    Comm_T01_T01W02 : ST_FB_30051_CommIn201;
    T01W01_Loaded : BOOL;
    T01W02_Loaded : BOOL;
END_VAR

(* Section T01W01: ladder, written here as Structured Text *)

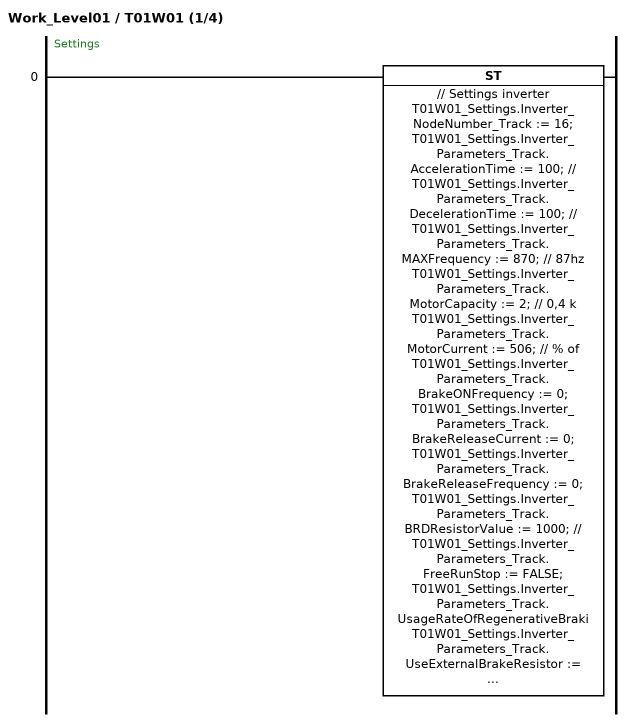
(* Rung 0: Settings *)
// Settings inverter
T01W01_Settings.Inverter_NodeNumber_Track := 16;
T01W01_Settings.Inverter_Parameters_Track.AccelerationTime := 100; // 1 sec
T01W01_Settings.Inverter_Parameters_Track.DecelerationTime := 100; // 1 sec
T01W01_Settings.Inverter_Parameters_Track.MAXFrequency := 870; // 87hz
T01W01_Settings.Inverter_Parameters_Track.MotorCapacity := 2; // 0,4 kw
T01W01_Settings.Inverter_Parameters_Track.MotorCurrent := 506; // % of maximum
T01W01_Settings.Inverter_Parameters_Track.BrakeONFrequency := 0;
T01W01_Settings.Inverter_Parameters_Track.BrakeReleaseCurrent := 0;
T01W01_Settings.Inverter_Parameters_Track.BrakeReleaseFrequency := 0;
T01W01_Settings.Inverter_Parameters_Track.BRDResistorValue := 1000; // = 100,0 ohm, this is the minimum value
T01W01_Settings.Inverter_Parameters_Track.FreeRunStop := FALSE;
T01W01_Settings.Inverter_Parameters_Track.UsageRateOfRegenerativeBraking := 0;
T01W01_Settings.Inverter_Parameters_Track.UseExternalBrakeResistor := FALSE;

T01W01_Settings.MaxSpeed := 5000;
T01W01_Settings.MinSpeed := 3500;
T01W01_Settings.MAX_Run_Time := 1800;
T01W01_Settings.TimeDelayON_IS201 := 1;
T01W01_Settings.TimeDelayOFF_IS201:= 20;
T01W01_Settings.TimeDelayON_IS202 := 1;
T01W01_Settings.TimeDelayOFF_IS202 := 20;
T01W01_Settings.TimeDelayON_ISPresent := 10;
T01W01_Settings.TimeDelayOFF_ISPresent := 10;
T01W01_Settings.TimeDelayON_LSTrackDown := 20;
T01W01_Settings.TimeDelayON_LSTrackUp := 20;
T01W01_Settings.TrackDirection := T01W01_Direction;
T01W01_Settings.HardwareCodeBuffer:= 202;
T01W01_Settings.DoTransferInbound_101:= TRUE;
T01W01_Settings.DoTransferOutbound_101:= TRUE;
T01W01_Settings.DoTransferInbound_Buffer:= FALSE; // Must be false as soon as BoweryOS and Dat-A-Control 
T01W01_Settings.DoTransferOutbound_Buffer:= TRUE;
T01W01_Settings.DoubleSolenoidValve:= TRUE;

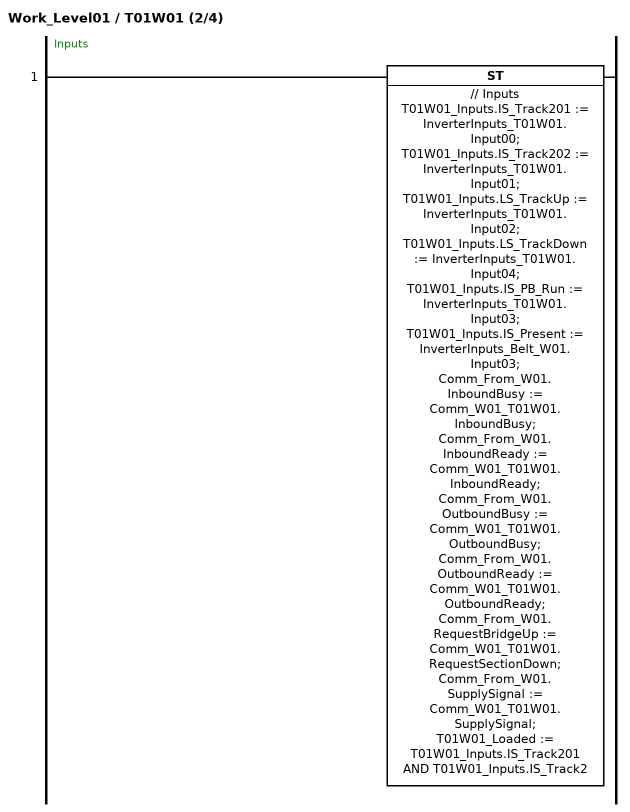
(* Rung 1: Inputs *)
// Inputs
T01W01_Inputs.IS_Track201 := InverterInputs_T01W01.Input00;
T01W01_Inputs.IS_Track202 := InverterInputs_T01W01.Input01;
T01W01_Inputs.LS_TrackUp := InverterInputs_T01W01.Input02;
T01W01_Inputs.LS_TrackDown := InverterInputs_T01W01.Input04;
T01W01_Inputs.IS_PB_Run := InverterInputs_T01W01.Input03;
T01W01_Inputs.IS_Present := InverterInputs_Belt_W01.Input03;

Comm_From_W01.InboundBusy := Comm_W01_T01W01.InboundBusy;
Comm_From_W01.InboundReady := Comm_W01_T01W01.InboundReady;
Comm_From_W01.OutboundBusy := Comm_W01_T01W01.OutboundBusy;
Comm_From_W01.OutboundReady := Comm_W01_T01W01.OutboundReady;
Comm_From_W01.RequestBridgeUp := Comm_W01_T01W01.RequestSectionDown;
Comm_From_W01.SupplySignal := Comm_W01_T01W01.SupplySignal;

T01W01_Loaded := T01W01_Inputs.IS_Track201 AND T01W01_Inputs.IS_Track202;

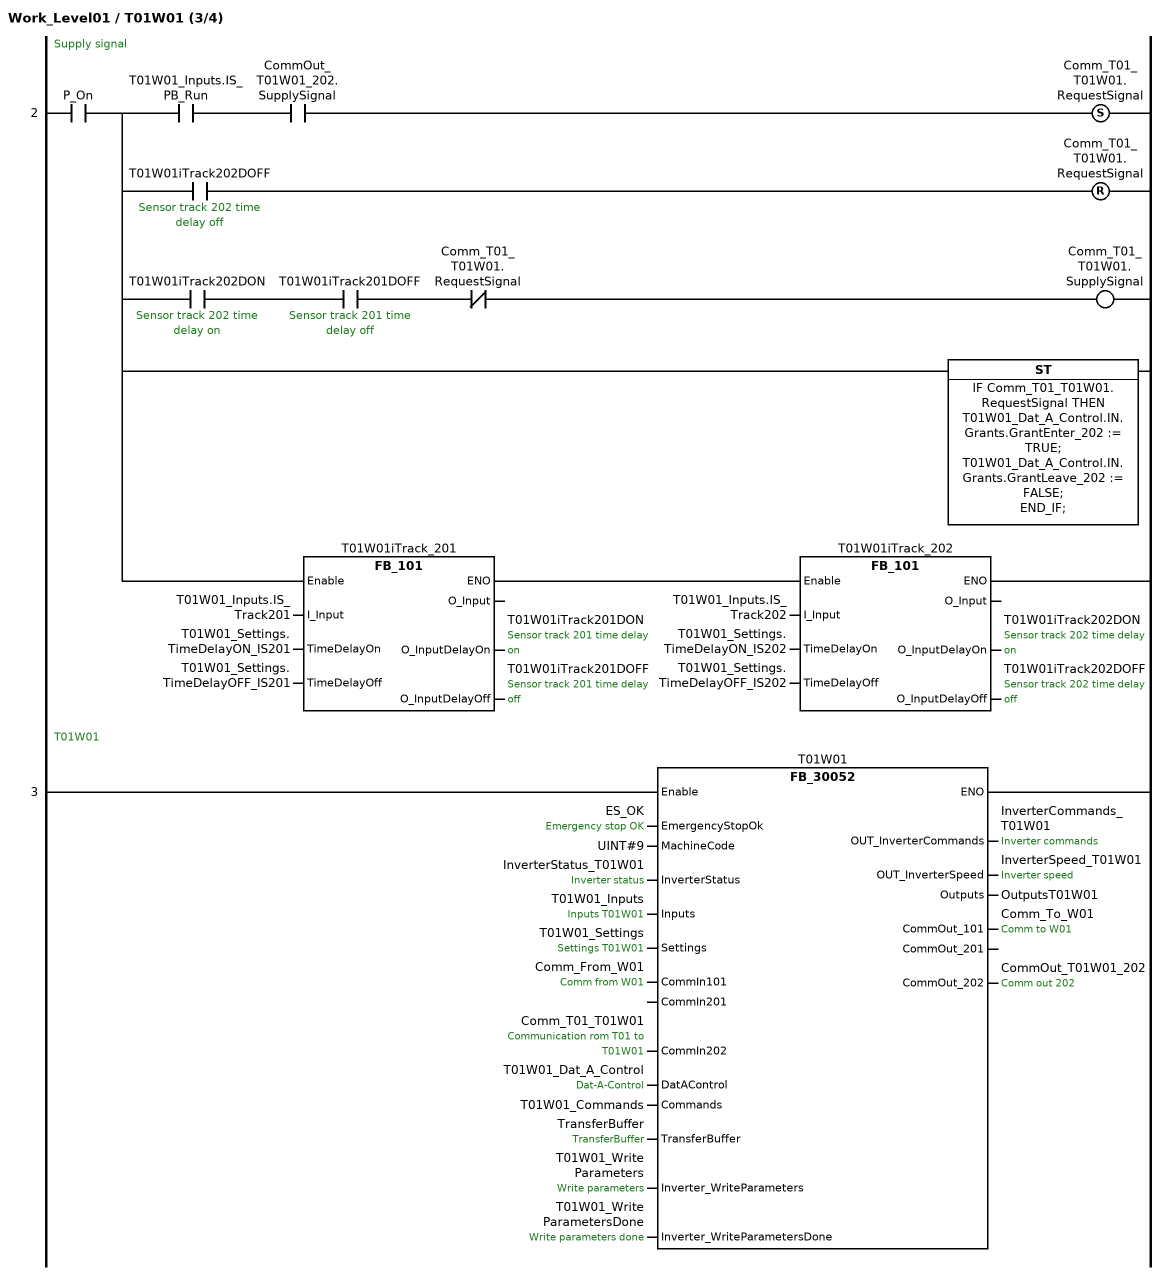
(* Rung 2: Supply signal *)
IF P_On AND T01W01_Inputs.IS_PB_Run AND CommOut_T01W01_202.SupplySignal THEN
    Comm_T01_T01W01.RequestSignal := TRUE;
END_IF;
IF P_On AND T01W01iTrack202DOFF THEN Comm_T01_T01W01.RequestSignal := FALSE; END_IF;
Comm_T01_T01W01.SupplySignal := P_On AND T01W01iTrack202DON AND T01W01iTrack201DOFF AND NOT Comm_T01_T01W01.RequestSignal;
IF P_On THEN
    IF Comm_T01_T01W01.RequestSignal THEN
    	T01W01_Dat_A_Control.IN.Grants.GrantEnter_202 := TRUE;
    	T01W01_Dat_A_Control.IN.Grants.GrantLeave_202 := FALSE;
    END_IF;
END_IF;
T01W01iTrack_201(Enable := P_On, I_Input := T01W01_Inputs.IS_Track201, TimeDelayOn := T01W01_Settings.TimeDelayON_IS201, TimeDelayOff := T01W01_Settings.TimeDelayOFF_IS201, O_InputDelayOn => T01W01iTrack201DON, O_InputDelayOff => T01W01iTrack201DOFF);
T01W01iTrack_202(Enable := T01W01iTrack_201.ENO, I_Input := T01W01_Inputs.IS_Track202, TimeDelayOn := T01W01_Settings.TimeDelayON_IS202, TimeDelayOff := T01W01_Settings.TimeDelayOFF_IS202, O_InputDelayOn => T01W01iTrack202DON, O_InputDelayOff => T01W01iTrack202DOFF);
(* Rung 3: T01W01 *)
T01W01(Enable := TRUE, EmergencyStopOk := ES_OK, MachineCode := UINT#9, InverterStatus := InverterStatus_T01W01, Inputs := T01W01_Inputs, Settings := T01W01_Settings, CommIn101 := Comm_From_W01, CommIn202 := Comm_T01_T01W01, DatAControl := T01W01_Dat_A_Control, Commands := T01W01_Commands, TransferBuffer := TransferBuffer, Inverter_WriteParameters := T01W01_WriteParameters, Inverter_WriteParametersDone := T01W01_WriteParametersDone, OUT_InverterCommands => InverterCommands_T01W01, OUT_InverterSpeed => InverterSpeed_T01W01, Outputs => OutputsT01W01, CommOut_101 => Comm_To_W01, CommOut_202 => CommOut_T01W01_202);

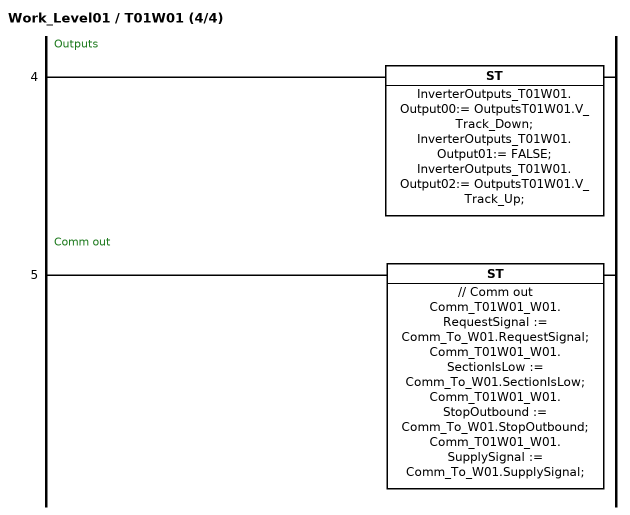
(* Rung 4: Outputs *)
InverterOutputs_T01W01.Output00:= OutputsT01W01.V_Track_Down;
InverterOutputs_T01W01.Output01:= FALSE;
InverterOutputs_T01W01.Output02:= OutputsT01W01.V_Track_Up;
(* Rung 5: Comm out *)
// Comm out
Comm_T01W01_W01.RequestSignal := Comm_To_W01.RequestSignal;
Comm_T01W01_W01.SectionIsLow := Comm_To_W01.SectionIsLow;
Comm_T01W01_W01.StopOutbound := Comm_To_W01.StopOutbound;
Comm_T01W01_W01.SupplySignal := Comm_To_W01.SupplySignal;

(* Section W01: ladder, written here as Structured Text *)

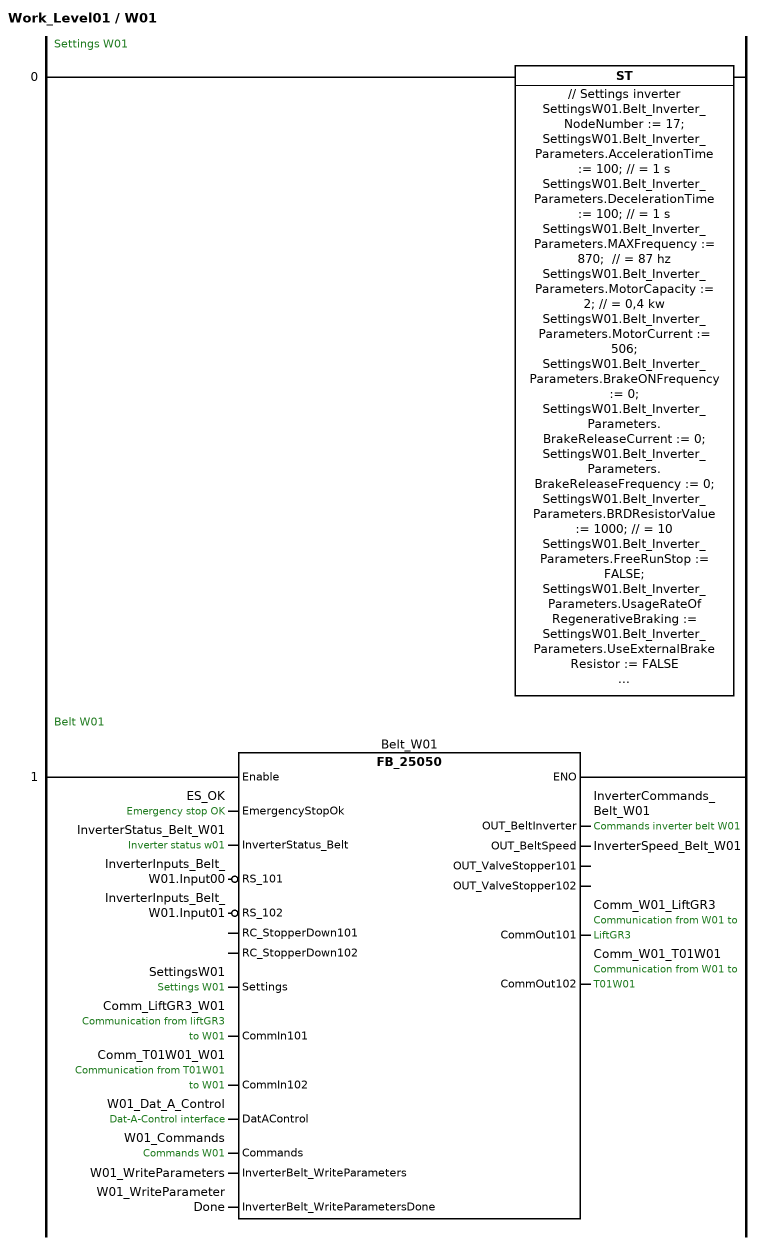
(* Rung 0: Settings W01 *)
// Settings inverter
SettingsW01.Belt_Inverter_NodeNumber := 17;
SettingsW01.Belt_Inverter_Parameters.AccelerationTime := 100; // = 1 second
SettingsW01.Belt_Inverter_Parameters.DecelerationTime := 100; // = 1 second
SettingsW01.Belt_Inverter_Parameters.MAXFrequency := 870;  // = 87 hz
SettingsW01.Belt_Inverter_Parameters.MotorCapacity := 2; // = 0,4 kw
SettingsW01.Belt_Inverter_Parameters.MotorCurrent := 506;
SettingsW01.Belt_Inverter_Parameters.BrakeONFrequency := 0;
SettingsW01.Belt_Inverter_Parameters.BrakeReleaseCurrent := 0;
SettingsW01.Belt_Inverter_Parameters.BrakeReleaseFrequency := 0;
SettingsW01.Belt_Inverter_Parameters.BRDResistorValue := 1000; // = 100,0 ohm, this is the minimum value
SettingsW01.Belt_Inverter_Parameters.FreeRunStop := FALSE;
SettingsW01.Belt_Inverter_Parameters.UsageRateOfRegenerativeBraking := 0;
SettingsW01.Belt_Inverter_Parameters.UseExternalBrakeResistor := FALSE;

SettingsW01.Belt_Max_Run_Time := 1800;
SettingsW01.Belt_Speed_Max := 5300;
SettingsW01.Belt_Speed_Min :=3500;
SettingsW01.Belt_Speed_Outbound101 := 4600;
SettingsW01.Belt_Speed_Outbound102 := 5000;
SettingsW01.TimeDelayOFF_RS101 := 10;
SettingsW01.TimeDelayON_RS101 := 10;
SettingsW01.TimeDelayOFF_RS102 := 10;
SettingsW01.TimeDelayON_RS102 := 10;
SettingsW01.Time_Belt_Fast := 170;
SettingsW01.DoNotCheckSensors := TRUE;
SettingsW01.NoInstructionInbound101 := TRUE;
SettingsW01.NoInstructionInbound102 := FALSE;
(* Rung 1: Belt W01 *)
Belt_W01(Enable := TRUE, EmergencyStopOk := ES_OK, InverterStatus_Belt := InverterStatus_Belt_W01, RS_101 := NOT InverterInputs_Belt_W01.Input00, RS_102 := NOT InverterInputs_Belt_W01.Input01, Settings := SettingsW01, CommIn101 := Comm_LiftGR3_W01, CommIn102 := Comm_T01W01_W01, DatAControl := W01_Dat_A_Control, Commands := W01_Commands, InverterBelt_WriteParameters := W01_WriteParameters, InverterBelt_WriteParametersDone := W01_WriteParameterDone, OUT_BeltInverter => InverterCommands_Belt_W01, OUT_BeltSpeed => InverterSpeed_Belt_W01, CommOut101 => Comm_W01_LiftGR3, CommOut102 => Comm_W01_T01W01);

(* Section T01W02: ladder, written here as Structured Text *)

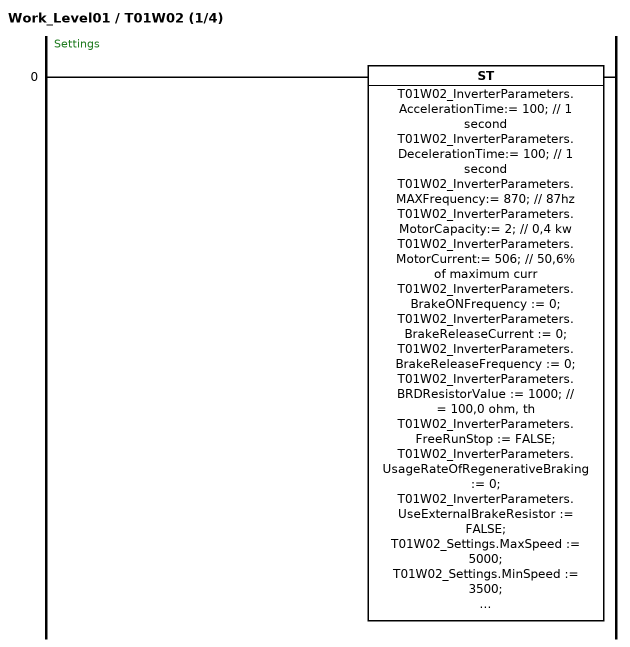
(* Rung 0: Settings *)
T01W02_InverterParameters.AccelerationTime:= 100; // 1 second
T01W02_InverterParameters.DecelerationTime:= 100; // 1 second
T01W02_InverterParameters.MAXFrequency:= 870; // 87hz
T01W02_InverterParameters.MotorCapacity:= 2; // 0,4 kw
T01W02_InverterParameters.MotorCurrent:= 506; // 50,6% of maximum current
T01W02_InverterParameters.BrakeONFrequency := 0;
T01W02_InverterParameters.BrakeReleaseCurrent := 0;
T01W02_InverterParameters.BrakeReleaseFrequency := 0;
T01W02_InverterParameters.BRDResistorValue := 1000; // = 100,0 ohm, this is the minimum value
T01W02_InverterParameters.FreeRunStop := FALSE;
T01W02_InverterParameters.UsageRateOfRegenerativeBraking := 0;
T01W02_InverterParameters.UseExternalBrakeResistor := FALSE;

T01W02_Settings.MaxSpeed := 5000;
T01W02_Settings.MinSpeed := 3500;
T01W02_Settings.MAX_Run_Time := 1800;
T01W02_Settings.TimeDelayON_IS201 := 1;
T01W02_Settings.TimeDelayOFF_IS201:= 20;
T01W02_Settings.TimeDelayON_IS202 := 1;
T01W02_Settings.TimeDelayOFF_IS202 := 20;
T01W02_Settings.TimeDelayON_ISPresent := 10;
T01W02_Settings.TimeDelayOFF_ISPresent := 10;
T01W02_Settings.TimeDelayON_LSTrackDown := 20;
T01W02_Settings.TimeDelayON_LSTrackUp := 20;
T01W02_Settings.TrackDirection := T01W02_Direction;
T01W02_Settings.HardwareCodeBuffer:= 201;
T01W02_Settings.DoTransferInbound_101:= TRUE;
T01W02_Settings.DoTransferOutbound_101:= TRUE;
T01W02_Settings.DoTransferInbound_Buffer:= FALSE; // Must be false as soon as BoweryOS and Dat-A-Control
T01W02_Settings.DoTransferOutbound_Buffer:= TRUE;  
T01W02_Settings.DoubleSolenoidValve:= FALSE;

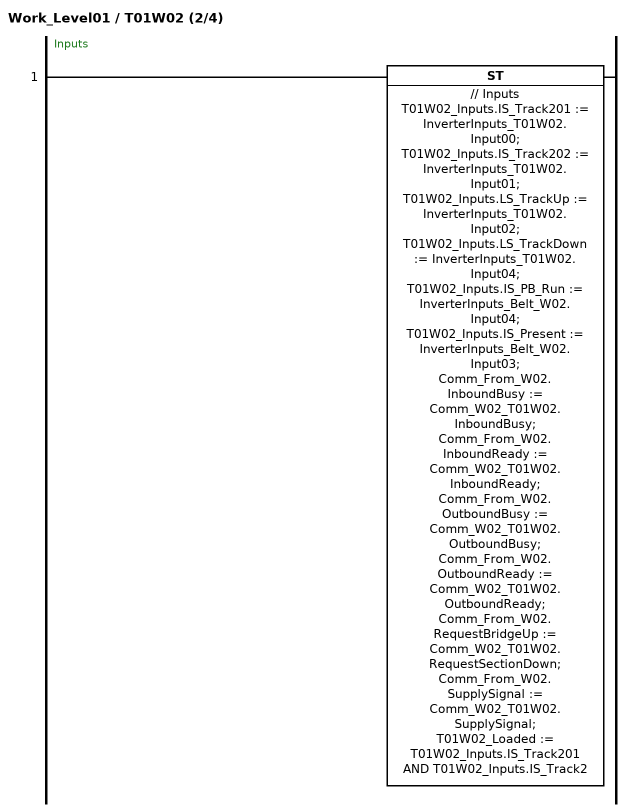
(* Rung 1: Inputs *)
// Inputs
T01W02_Inputs.IS_Track201 := InverterInputs_T01W02.Input00;
T01W02_Inputs.IS_Track202 := InverterInputs_T01W02.Input01;
T01W02_Inputs.LS_TrackUp := InverterInputs_T01W02.Input02;
T01W02_Inputs.LS_TrackDown := InverterInputs_T01W02.Input04;
T01W02_Inputs.IS_PB_Run := InverterInputs_Belt_W02.Input04;
T01W02_Inputs.IS_Present := InverterInputs_Belt_W02.Input03;

Comm_From_W02.InboundBusy := Comm_W02_T01W02.InboundBusy;
Comm_From_W02.InboundReady := Comm_W02_T01W02.InboundReady;
Comm_From_W02.OutboundBusy := Comm_W02_T01W02.OutboundBusy;
Comm_From_W02.OutboundReady := Comm_W02_T01W02.OutboundReady;
Comm_From_W02.RequestBridgeUp := Comm_W02_T01W02.RequestSectionDown;
Comm_From_W02.SupplySignal := Comm_W02_T01W02.SupplySignal;

T01W02_Loaded := T01W02_Inputs.IS_Track201 AND T01W02_Inputs.IS_Track202;

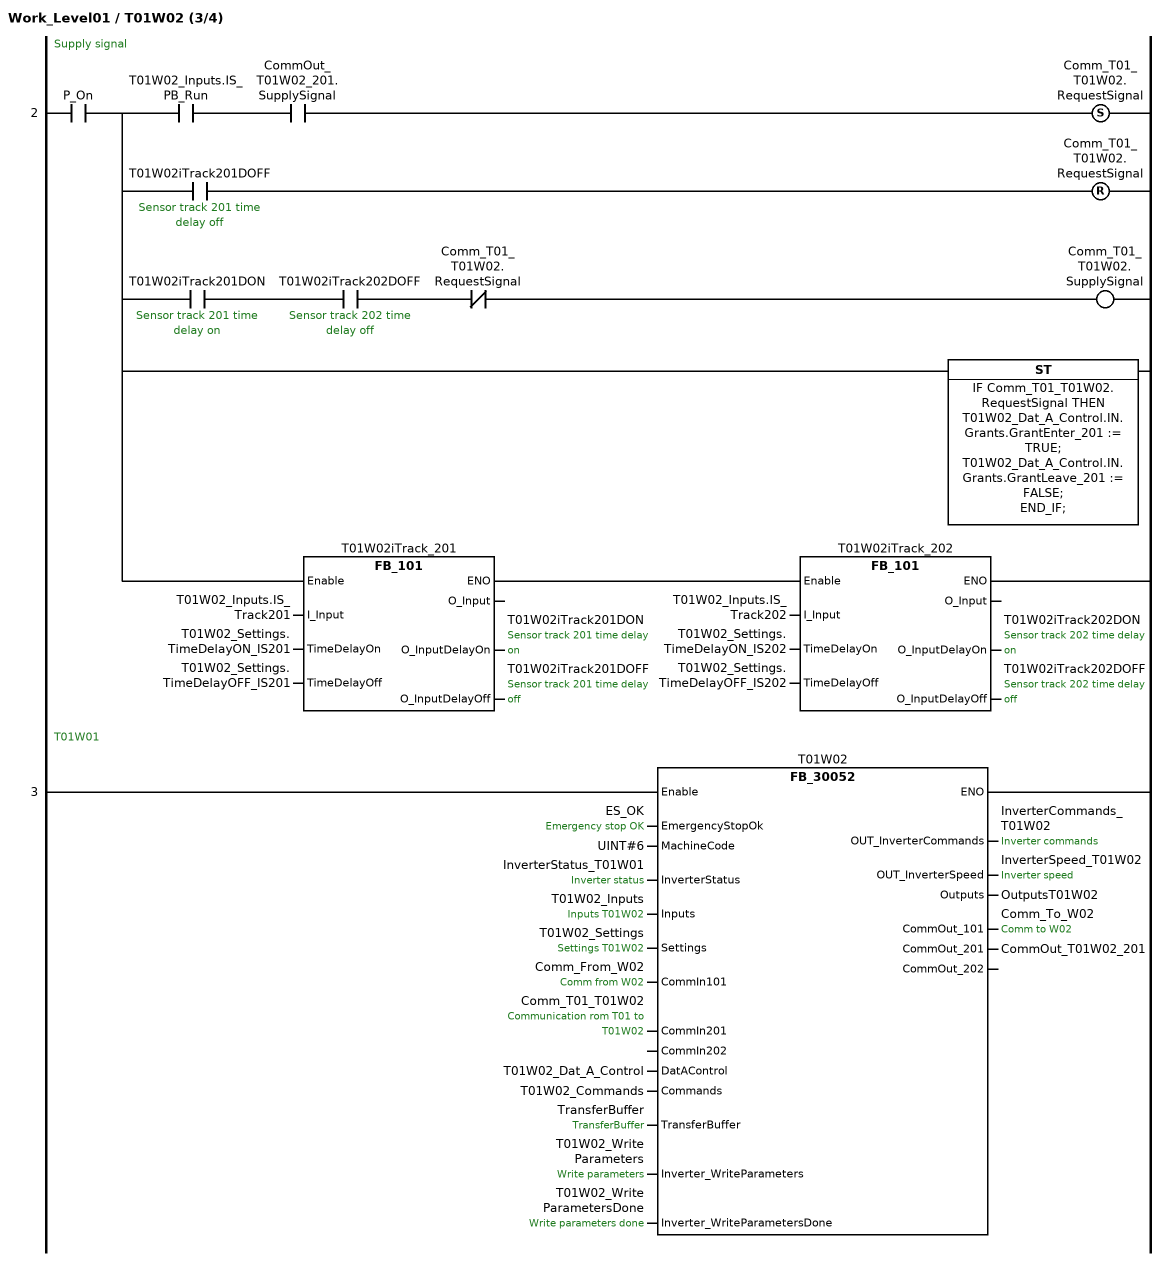
(* Rung 2: Supply signal *)
IF P_On AND T01W02_Inputs.IS_PB_Run AND CommOut_T01W02_201.SupplySignal THEN
    Comm_T01_T01W02.RequestSignal := TRUE;
END_IF;
IF P_On AND T01W02iTrack201DOFF THEN Comm_T01_T01W02.RequestSignal := FALSE; END_IF;
Comm_T01_T01W02.SupplySignal := P_On AND T01W02iTrack201DON AND T01W02iTrack202DOFF AND NOT Comm_T01_T01W02.RequestSignal;
IF P_On THEN
    IF Comm_T01_T01W02.RequestSignal THEN
    	T01W02_Dat_A_Control.IN.Grants.GrantEnter_201 := TRUE;
    	T01W02_Dat_A_Control.IN.Grants.GrantLeave_201 := FALSE;
    END_IF;
END_IF;
T01W02iTrack_201(Enable := P_On, I_Input := T01W02_Inputs.IS_Track201, TimeDelayOn := T01W02_Settings.TimeDelayON_IS201, TimeDelayOff := T01W02_Settings.TimeDelayOFF_IS201, O_InputDelayOn => T01W02iTrack201DON, O_InputDelayOff => T01W02iTrack201DOFF);
T01W02iTrack_202(Enable := T01W02iTrack_201.ENO, I_Input := T01W02_Inputs.IS_Track202, TimeDelayOn := T01W02_Settings.TimeDelayON_IS202, TimeDelayOff := T01W02_Settings.TimeDelayOFF_IS202, O_InputDelayOn => T01W02iTrack202DON, O_InputDelayOff => T01W02iTrack202DOFF);
(* Rung 3: T01W01 *)
T01W02(Enable := TRUE, EmergencyStopOk := ES_OK, MachineCode := UINT#6, InverterStatus := InverterStatus_T01W01, Inputs := T01W02_Inputs, Settings := T01W02_Settings, CommIn101 := Comm_From_W02, CommIn201 := Comm_T01_T01W02, DatAControl := T01W02_Dat_A_Control, Commands := T01W02_Commands, TransferBuffer := TransferBuffer, Inverter_WriteParameters := T01W02_WriteParameters, Inverter_WriteParametersDone := T01W02_WriteParametersDone, OUT_InverterCommands => InverterCommands_T01W02, OUT_InverterSpeed => InverterSpeed_T01W02, Outputs => OutputsT01W02, CommOut_101 => Comm_To_W02, CommOut_201 => CommOut_T01W02_201);

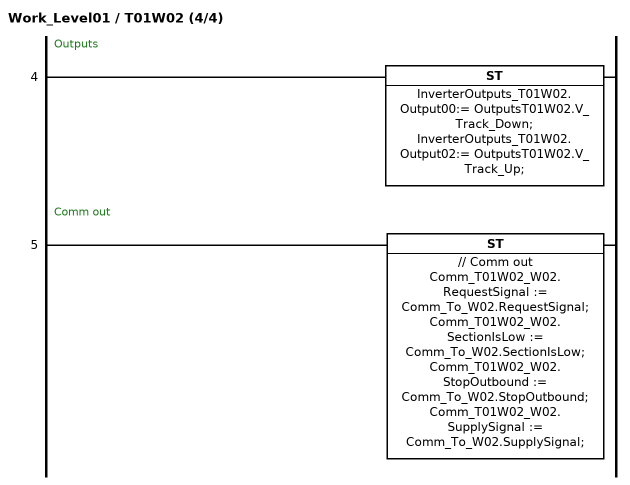
(* Rung 4: Outputs *)
InverterOutputs_T01W02.Output00:= OutputsT01W02.V_Track_Down;
InverterOutputs_T01W02.Output02:= OutputsT01W02.V_Track_Up;
(* Rung 5: Comm out *)
// Comm out
Comm_T01W02_W02.RequestSignal := Comm_To_W02.RequestSignal;
Comm_T01W02_W02.SectionIsLow := Comm_To_W02.SectionIsLow;
Comm_T01W02_W02.StopOutbound := Comm_To_W02.StopOutbound;
Comm_T01W02_W02.SupplySignal := Comm_To_W02.SupplySignal;

(* Section W02: ladder, written here as Structured Text *)

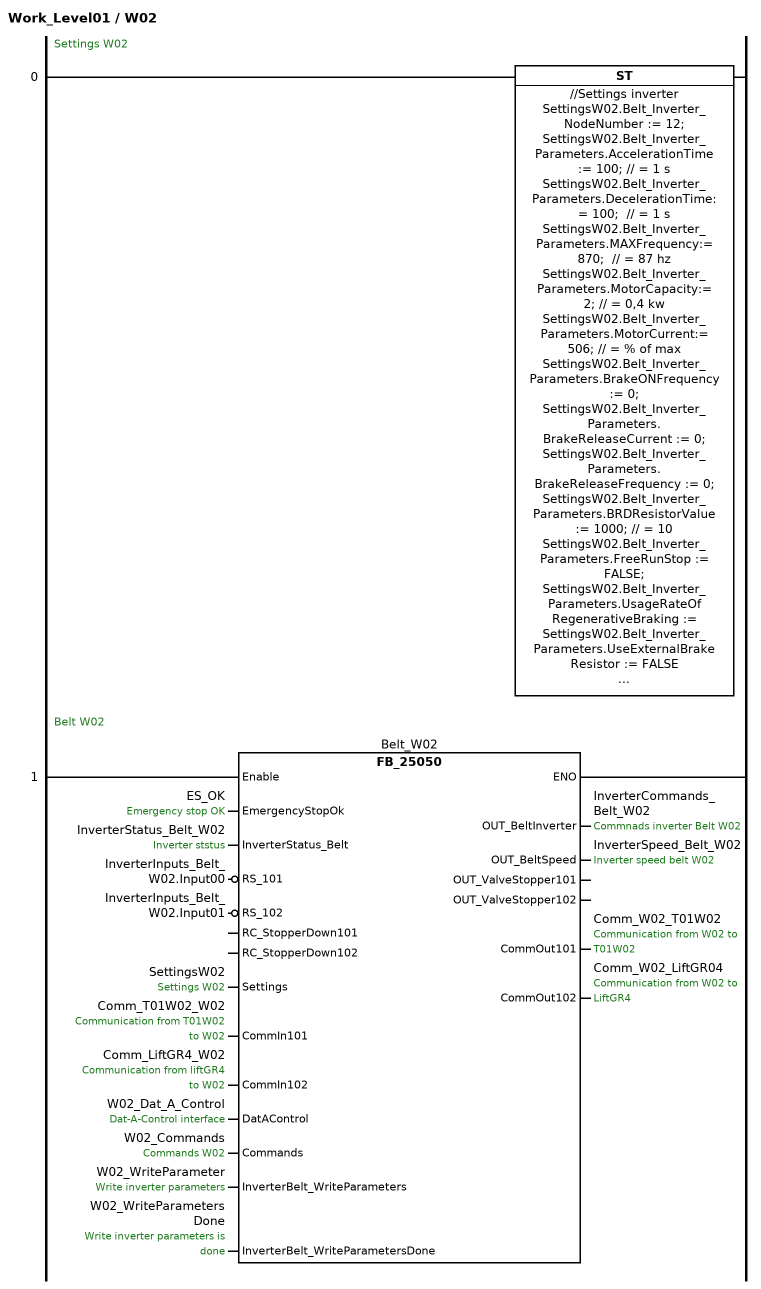
(* Rung 0: Settings W02 *)
//Settings inverter
SettingsW02.Belt_Inverter_NodeNumber := 12;
SettingsW02.Belt_Inverter_Parameters.AccelerationTime := 100; // = 1 second
SettingsW02.Belt_Inverter_Parameters.DecelerationTime:= 100;  // = 1 second
SettingsW02.Belt_Inverter_Parameters.MAXFrequency:= 870;  // = 87 hz
SettingsW02.Belt_Inverter_Parameters.MotorCapacity:= 2; // = 0,4 kw
SettingsW02.Belt_Inverter_Parameters.MotorCurrent:= 506; // = % of maximum current
SettingsW02.Belt_Inverter_Parameters.BrakeONFrequency := 0;
SettingsW02.Belt_Inverter_Parameters.BrakeReleaseCurrent := 0;
SettingsW02.Belt_Inverter_Parameters.BrakeReleaseFrequency := 0;
SettingsW02.Belt_Inverter_Parameters.BRDResistorValue := 1000; // = 100,0 ohm, this is the minimum value
SettingsW02.Belt_Inverter_Parameters.FreeRunStop := FALSE;
SettingsW02.Belt_Inverter_Parameters.UsageRateOfRegenerativeBraking := 0;
SettingsW02.Belt_Inverter_Parameters.UseExternalBrakeResistor := FALSE;

SettingsW02.Belt_Max_Run_Time:= 1800;
SettingsW02.Belt_Speed_Max := 5300;
SettingsW02.Belt_Speed_Min := 3500;
SettingsW02.Belt_Speed_Outbound101:= 5000;
SettingsW02.Belt_Speed_Outbound102 := 4600;
SettingsW02.TimeDelayOFF_RS101:= 10;
SettingsW02.TimeDelayON_RS101:= 10;
SettingsW02.TimeDelayOFF_RS102:= 10;
SettingsW02.TimeDelayON_RS102:= 10;
SettingsW02.Time_Belt_Fast := 170;
SettingsW02.DoNotCheckSensors:=TRUE;
SettingsW02.NoInstructionInbound101:= FALSE;
SettingsW02.NoInstructionInbound102:= TRUE;
(* Rung 1: Belt W02 *)
Belt_W02(Enable := TRUE, EmergencyStopOk := ES_OK, InverterStatus_Belt := InverterStatus_Belt_W02, RS_101 := NOT InverterInputs_Belt_W02.Input00, RS_102 := NOT InverterInputs_Belt_W02.Input01, Settings := SettingsW02, CommIn101 := Comm_T01W02_W02, CommIn102 := Comm_LiftGR4_W02, DatAControl := W02_Dat_A_Control, Commands := W02_Commands, InverterBelt_WriteParameters := W02_WriteParameter, InverterBelt_WriteParametersDone := W02_WriteParametersDone, OUT_BeltInverter => InverterCommands_Belt_W02, OUT_BeltSpeed => InverterSpeed_Belt_W02, CommOut101 => Comm_W02_T01W02, CommOut102 => Comm_W02_LiftGR04);
END_PROGRAM

PROGRAM Work_Mezzanine
VAR
    Belt_W06 : FB_25050;
    SettingsW06 : ST_FB_25050\Settings;  (* Settings W06 *)
    W06_WriteParameters : BOOL;  (* Write parameters to inverter *)
    W06_WriteParametersDone : BOOL;  (* Write parameters done *)
    SettingsW02 : ST_FB_25050\Settings;  (* Settings W02 *)
    Belt_W07 : FB_25050;
    SettingsW07 : ST_FB_25050\Settings;  (* Settings W07 *)
    W07_WriteParameters : BOOL;  (* Write inverter parameters *)
    W07_WriteParametersDone : BOOL;  (* Write inverter parameters done *)
    SettingsW01 : ST_FB_25050\Settings;  (* Settings W01 *)
    T02W07 : FB_30051;
    WriteParametersBelt_T02W07 : BOOL;  (* Write parameters *)
    WriteParametersTrack_T02W07 : BOOL;  (* Write parameters *)
    Write : BOOL;
    WriteParametersBeltDone_T02W07 : BOOL;  (* Write parameters done *)
    WriteParametersTrackDone_T02W07 : BOOL;  (* Write parameters done *)
    SettingsT02W07 : ST_FB_30051_Settings;  (* Settings T02W07 *)
    InputsT02W07 : ST_FB_30051_Inputs;  (* Inputs T02W07 *)
    OutputsT02W07 : ST_FB_30051_Outputs;  (* Outputs T02W07 *)
    T02W06 : FB_30051;
    InputsT02W06 : ST_FB_30051_Inputs;  (* INputs T02W06 *)
    SettingsT02W06 : ST_FB_30051_Settings;  (* Settings T02W06 *)
    WriteParametersBelt_T02W06 : BOOL;  (* Write parameters *)
    WriteParametersTrack_T02W06 : BOOL;  (* Write parameters *)
    WriteParametersBeltDone_T02W06 : BOOL;  (* Write parameters done *)
    WriteParametersTrackDone_T02W06 : BOOL;  (* Write parameters done *)
    OutputsT02W06 : ST_FB_30051_Outputs;  (* Outputs T02W06 *)
    Comm_From_W06 : ST_Comm_Pipe_To_Track;  (* communication from W06 *)
    Comm_To_W06 : ST_Comm_Track_To_Pipe;  (* Communication to W06 *)
    Comm_From_W07 : ST_Comm_Pipe_To_Track;  (* Communication from W07 *)
    Comm_To_W07 : ST_Comm_Track_To_Pipe;  (* Communication to W07 *)
    IS_201_Stacker : FB_101;
    I_201_Stacker : BOOL;  (* input 201 *)
    I_201_StackerDON : BOOL;  (* input 201 stacker delay on *)
    I_201_StackerDOFF : BOOL;  (* input 201 stacker delay off *)
    IS_202_Stacker : FB_101;
    I_202_Stacker : BOOL;  (* input 202 *)
    I_202_StackerDON : BOOL;  (* INput 202 stacker delay on *)
    I_202_StackerDOFF : BOOL;  (* Input 202 stacker delay off *)
    IS_StackerEmpty : FB_101;
    I_StackerEmpty : BOOL;  (* stacker empty *)
    IS_StackerFull : FB_101;
    I_StackerFull : BOOL;  (* Stacker is full *)
    I_StackerEmptyDON : BOOL;  (* Stacker empty delay on *)
    I_StackerFullDON : BOOL;  (* Stacker full delay on *)
    IS_TrayAtPosition : FB_101;
    I_TrayAtPosition : BOOL;  (* Tray is at position *)
    RF_FreeUnderTray : FB_101;
    I_FreeUnderTray : BOOL;  (* Space free under tray *)
    RF_TrayPresent : FB_101;
    I_TrayPresent_Stacker : BOOL;  (* Tray present in stacker *)
    I_FreeUnderTray_Stacker : BOOL;  (* Space free under tray *)
    I_FreeUnderTrayDON : BOOL;  (* Space free under tray delay on *)
    I_TrayPresent_StackerDON : BOOL;  (* Tray present in stacker delay on *)
    Motor_Track_Stacker : FB_1011;
    Track_Stacker_Ref_Rev : BOOL;  (* Motor reference is reverse *)
    Track_Stacker_Ref_Fwd : BOOL;  (* Motor reference is forward *)
    Track_Stacker_ConditionsGlobal : BOOL;  (* Global conditions ok *)
    Track_Stacker_ConditionsFwd : BOOL;  (* Forward conditions ok *)
    Track_Stacker_ConditionsRev : BOOL;  (* Reverse conditions ok *)
    Stacker_MachineMode : ST_MachineMode;  (* Stacker machine mode *)
    Track_Stacker_FWD : BOOL;  (* Track stacker forward *)
    Track_Stacker_REV : BOOL;  (* Track_Stacker_REV *)
END_VAR
VAR RETAIN
    Stacker_Cyc_Load : ST_Stacker_Cyc_Load;  (* cycle load; Step00 Instruction is load a tray; Step01 Supply signal present, dot transfer; Step02 Transfer OK; Step03 Tray is present at section, check stack full; Step04 Stack is not full, move stacker up; Step05 Tray is lifted, do transfer; Step06 Tray is lifted, do transfer; Step08 Stack is full, reset cycle; Step07 Transfer OK, reset cycle *)
    Stacker_Cyc_Unload : ST_Stacker_Cyc_Unload;  (* Cycle unload; Step00 Instruction is to unload tray; Step01 Tray is present in stacker, start move down; Step02 Tray is going down; Step03 Tray is at the track; Step04 Transfer is ok, reset cycle; Step05 Error tray not detected at track *)
END_VAR
VAR
    Track_Stacker_Speed_Ref : INT;  (* Speed reference *)
    Inverter_Track_Stacker : FB_305;
    Track_Stacker_Parameters : ST_MX2\Parameters;  (* Track stacker parameters *)
    Track_Stacker_WriteParameters : BOOL;  (* write parameters *)
    Track_Stacker_WriteParametersDone : BOOL;  (* Write parameters done *)
    Stacker_ConditionsGlobal : BOOL;  (* Global conditions ok *)
    Stacker_ConditionsUp : BOOL;  (* conditions up ok *)
    Stacker_ConditionsDown : BOOL;  (* Conditions down ok *)
    Motor_Stacker : FB_1011;
    Stacker_Ref_Up : BOOL;  (* Stacker reference is up *)
    Stacker_Ref_Down : BOOL;  (* Stacker reference is down *)
    Stacker_TotalDone : UDINT;
    M_Stacker_Up : BOOL;  (* Motor stacker up *)
    M_Stacker_Down : BOOL;  (* Motor stacker down *)
    Stacker_Speed_Ref : INT;  (* Stacker speed reference *)
    INverter_Stacker : FB_305;
    Stacker_Parameters : ST_MX2\Parameters;  (* Stacker inverter parameters *)
    Stacker_WriteParameters : BOOL;  (* Write parameters *)
    Stacker_WriteParametersDone : BOOL;  (* Write parameters done *)
    Stacker_Instructions : FB_904;
    Stacker_InstructionParameters : ST_Instruction_Conditions_Standaard;  (* Instruction parameters *)
    Stacker_StartInstruction : BOOL;  (* Start instruction *)
    Stacker_LoadGate : UINT;  (* Load gate *)
    Stacker_UnloadGate : UINT;  (* Unload gate *)
    Stacker_ResetAlarm : BOOL;  (* Reset alarm *)
    Stacker_ResetCycle : BOOL;  (* Reset cycle *)
    TransferOK : BOOL;  (* Transfer ok *)
    Comm_Stacker_T02W07 : ST_Comm_Track_To_Track;  (* Communication from stacker *)
    Comm_T02W07_Stacker : ST_Comm_Track_To_Track;  (* Communication to stacker *)
    hulp1 : BOOL;
    hulp2 : BOOL;
    hulp3 : BOOL;
    hulp4 : BOOL;
    Semi_Automatic_Stacker : FB_307;
    Stacker : BOOL;
    StackerStop_SA : BOOL;  (* Stacker stop in semi automatic *)
    Stacker_SA_Up : BOOL;  (* Stacker semi automatic up *)
    STacker_SA_Down : BOOL;  (* Stacker semi automatic down *)
    Semi_Automatic_Stacker_Track : FB_307;
    StackerTrack_SA_FWD : BOOL;  (* Stacker track semi automatic forward *)
    StackerTrack_SA_REV : BOOL;  (* Stacker track semi automatic reverse *)
    I_TrayAtPositionDON : BOOL;  (* Tray at poition delay on *)
    Comm_T02_T02W07 : ST_Comm_Track_To_Track;  (* Communication from T02 *)
    Comm_T02W07_T02 : ST_Comm_Track_To_Track;  (* Communication to T02 *)
    Comm_T02_T02W06 : ST_Comm_Track_To_Track;  (* Communication from T02 *)
    Comm_T02W06_T02 : ST_Comm_Track_To_Track;  (* Communicatio to T02 *)
    TimerStackerBoost : _sTimer;  (* Timer stacker boost *)
    W07_RC_StoppersDown101 : BOOL;  (* HelpBit to combine inputs *)
    W06_RC_StoppersDown101 : BOOL;
    W06_RC_StoppersDown102 : BOOL;  (* Helpbit to combite inputs *)
    HB_T02W06_TransferOK : BOOL;
    PB_EjectTray : FB_101;
    I_PB_EjectTray : BOOL;  (* Push button to eject tray from stacker *)
    I_PB_EjectTrayDON : BOOL;  (* Push button to eject tray from stacker Delayed On *)
    I_PB_EjectTrayDOFF : BOOL;  (* Push button to eject tray from stacker delayed off *)
    PB_InsertTray : FB_101;
    I_PB_InsertTray : BOOL;  (* Pushbutton to instert tray into Stacker *)
    I_PB_InstertTrayDON : BOOL;  (* Pushbutton to instert tray into Stacker Delayed ON *)
    I_PB_InsertTrayDOFF : BOOL;  (* Pushbutton to instert tray into Stacker Delayed OFF *)
    Stacker_C : BOOL;
    Stacker_AtPositionTimer : UINT;  (* Settig timer input timer *)
    Track201DON : BOOL;  (* Sensor track 201 time delay on *)
    Track201DOFF : BOOL;  (* Sensor track 201 time delay off *)
    TRack_201 : FB_101;
    TRack_202 : FB_101;
    Track202DON : BOOL;  (* Sensor track 202 time delay on *)
    Track202DOFF : BOOL;  (* Sensor track 202 time delay off *)
    T02W06iTrack_201 : FB_101;
    T02W06iTrack201DON : BOOL;  (* Sensor track 201 time delay on *)
    T02W06iTrack201DOFF : BOOL;  (* Sensor track 201 time delay off *)
    T0W06iTrack_202 : FB_101;
    T02W06iTrack202DON : BOOL;  (* Sensor track 202 time delay on *)
    T02W06iTrack202DOFF : BOOL;  (* Sensor track 202 time delay off *)
    T02W07iTrack_201 : FB_101;
    T02W07iTrack201DON : BOOL;  (* Sensor track 201 time delay on *)
    T02W07iTrack201DOFF : BOOL;  (* Sensor track 201 time delay off *)
    T0W07iTrack_202 : FB_101;
    T02W07iTrack202DON : BOOL;  (* Sensor track 202 time delay on *)
    T02W07iTrack202DOFF : BOOL;  (* Sensor track 202 time delay off *)
    Stacker_BrakeReleaseFreq : INT;  (* Minimum frequenty befoe release brake *)
    Stacker_BoostTime : UINT;  (* Time for boost up/down *)
    Berke_TEST : BOOL;
END_VAR
VAR_EXTERNAL
    Dummy : BOOL;
    ES_OK : BOOL;
    InverterStatus_W06 : ST_MX2\Status;
    InverterInputs_W06 : ST_MX2\Input;
    Comm_T02W06_W06 : ST_FB_25050\CommInPipe;  (* Communication from T02W06 to W06 *)
    Comm_LiftGR3_W06 : ST_FB_25050\CommInPipe;  (* Communication from lift GR03 to W06 *)
    InverterCommands_W06 : ST_MX2\Command;  (* Inverter commands *)
    InverterSpeed_W06 : INT;  (* Inverter speed *)
    Comm_W06_T02W06 : ST_FB_25050\CommOutPipe;  (* Communication from W06 to T02W06 *)
    Comm_W06_LiftGR3 : ST_FB_25050\CommOutPipe;  (* Communication from W06 to LiftGR3 *)
    InverterStatus_W07 : ST_MX2\Status;  (* Inverter status W07 *)
    InverterInputs_W07 : ST_MX2\Input;
    InverterCommands_W07 : ST_MX2\Command;  (* Inverter commands *)
    InverterSpeed_W07 : INT;  (* Inverter speed *)
    Comm_W07_T02W07 : ST_FB_25050\CommOutPipe;  (* Communication from W07 to T02W07 *)
    Comm_W07_LiftGR04 : ST_FB_25050\CommOutPipe;  (* Communication from W07 to LiftGR04 *)
    W07_Dat_A_Control : ST_DatAControl_Standard;  (* Dat a control interface *)
    W07_Commands : ST_FB_25050\Commands;  (* Comands W07 *)
    Comm_LiftGR4_W07 : ST_FB_25050\CommInPipe;  (* Communication from lift GR04 to W07 *)
    Comm_T02W07_W07 : ST_FB_25050\CommInPipe;  (* Communication from T02W07 to W07 *)
    W06_Dat_A_Control : ST_DatAControl_Standard;  (* Dat a control interface *)
    W06_Commands : ST_FB_25050\Commands;  (* Commands W06 *)
    TransferBuffer : ST_TransferBuffer;
    T02W07_DatAControl : ST_DatAControl_Standard;  (* Dat a Control *)
    T02W07_Commands : ST_FB_30051_Commands;  (* Commands *)
    InverterStatus_T02W07 : ST_MX2\Status;  (* Inverter status *)
    InverterStatus_T02W07_Belt : ST_MX2\Status;  (* Inverter status *)
    InverterCommands_T02W07_Belt : ST_MX2\Command;  (* Inverter commands *)
    InverterCommands_T02W07 : ST_MX2\Command;  (* Inverter commands *)
    InverterSpeed_T02W07_Belt : INT;  (* inverter speed *)
    InverterSpeed_T02W07 : INT;  (* Inverter speed *)
    InverterStatus_T02W06_Belt : ST_MX2\Status;  (* Inverter status *)
    InverterStatus_T02W06 : ST_MX2\Status;  (* Inverter status *)
    InverterCommands_T02W06_Belt : ST_MX2\Command;  (* Inverter commands *)
    InverterCommands_T02W06 : ST_MX2\Command;  (* Inverter commands *)
    InverterSpeed_T02W06_Belt : INT;  (* Inverter speed *)
    InverterSpeed_T02W06 : INT;  (* Inverter speed *)
    T02W06_DatAControl : ST_DatAControl_Standard;  (* Datacontrol interface *)
    T02W06_Commands : ST_FB_30051_Commands;  (* Commands T02W06 *)
    InverterInputs_T02W07 : ST_MX2\Input;
    InverterInputs_T02W07_Belt : ST_MX2\Input;
    InverterOutputs_T02W07_Belt : ST_MX2\Output;
    InverterOutputs_T02W06_Belt : ST_MX2\Output;
    InverterInputs_T02W06 : ST_MX2\Input;
    InverterInputs_T02W06_Belt : ST_MX2\Input;
    InverterInputs_T02_Stacker : ST_MX2\Input;
    InverterInputs_Stacker : ST_MX2\Input;
    Stacker_DatAControl : ST_DatAControl_Standard;  (* Dat A Control; IN.MachineMode Machine mode; IN.Settings.ResetAlarm Reset alarm; OUT.Alarm01 Alarm 1; OUT.Alarm03 Alarm 3; IN.ManualMode Manual override *)
    Stacker_Commands : ST_Stacker_Commands;  (* Stacker commands; Track_Forward Track forward; Track_Reverse Track reverse; Track_Stop Stop track; StackerUp Commands stacker up; StackerDown Commands stacker up; StackerStop Command stop stacker *)
    InverterStatus_T02_Stacker : ST_MX2\Status;  (* Inverter status *)
    InverterCommands_T02_Stacker : ST_MX2\Command;  (* Inverter commands *)
    InverterSpeed_T02_Stacker : INT;  (* Inverter speed *)
    InverterStatus_Stacker : ST_MX2\Status;  (* Inverter status *)
    InverterCommands_Stacker : ST_MX2\Command;  (* Inverter commands *)
    InverterSpeed_Stacker : INT;  (* Inverter speed *)
    InverterOutputs_W07 : ST_MX2\Output;
    InverterOutputs_W06 : ST_MX2\Output;
    T02W07_Direction : UINT;
    T02W06_Direction : UINT;
    Supply_Stacker : BOOL;
    Insert_Stacker : BOOL;
    InverterOutputs_Stacker : ST_MX2\Output;
    T02W06_Loaded : BOOL;
    T02W07_Loaded : BOOL;
END_VAR
VAR
    _e1 : R_TRIG;
    _p2 : BOOL;
    _p3 : BOOL;
    _e4 : R_TRIG;
    _t5 : BOOL;
    _p6 : BOOL;
    _p7 : BOOL;
    _p8 : BOOL;
    _p9 : BOOL;
END_VAR

(* Section T02W06: ladder, written here as Structured Text *)

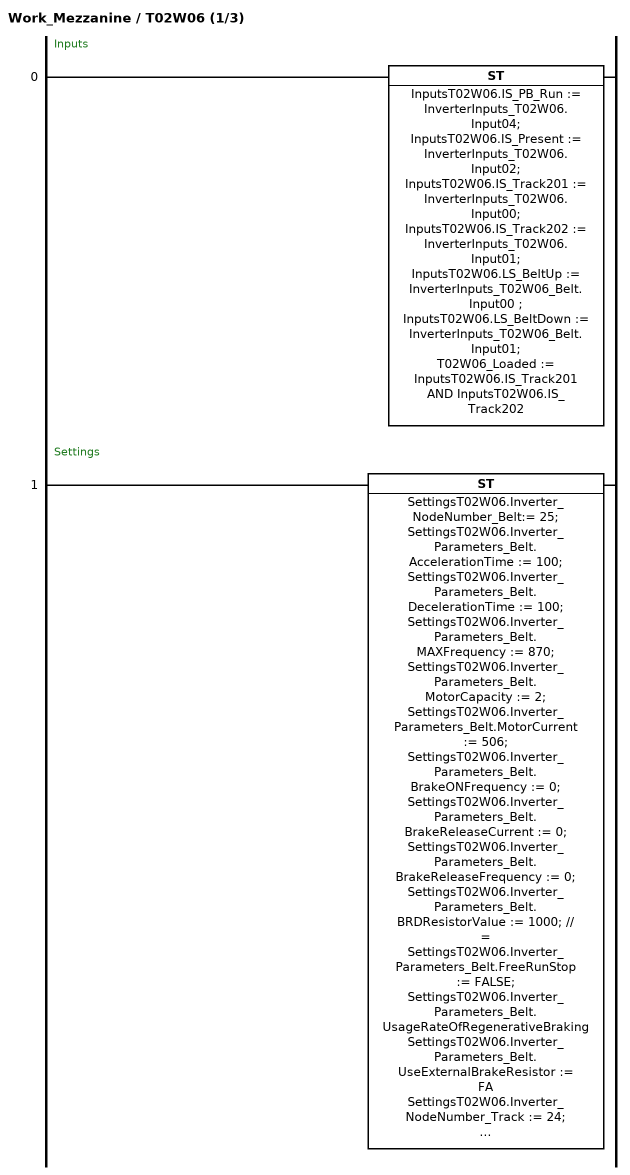
(* Rung 0: Inputs *)
InputsT02W06.IS_PB_Run := InverterInputs_T02W06.Input04;
InputsT02W06.IS_Present := InverterInputs_T02W06.Input02;
InputsT02W06.IS_Track201 := InverterInputs_T02W06.Input00;
InputsT02W06.IS_Track202 := InverterInputs_T02W06.Input01;
InputsT02W06.LS_BeltUp := InverterInputs_T02W06_Belt.Input00 ;
InputsT02W06.LS_BeltDown := InverterInputs_T02W06_Belt.Input01;

T02W06_Loaded := InputsT02W06.IS_Track201 AND InputsT02W06.IS_Track202;
(* Rung 1: Settings *)
SettingsT02W06.Inverter_NodeNumber_Belt:= 25;
SettingsT02W06.Inverter_Parameters_Belt.AccelerationTime := 100;
SettingsT02W06.Inverter_Parameters_Belt.DecelerationTime := 100;
SettingsT02W06.Inverter_Parameters_Belt.MAXFrequency := 870;
SettingsT02W06.Inverter_Parameters_Belt.MotorCapacity := 2;
SettingsT02W06.Inverter_Parameters_Belt.MotorCurrent := 506;
SettingsT02W06.Inverter_Parameters_Belt.BrakeONFrequency := 0;
SettingsT02W06.Inverter_Parameters_Belt.BrakeReleaseCurrent := 0;
SettingsT02W06.Inverter_Parameters_Belt.BrakeReleaseFrequency := 0;
SettingsT02W06.Inverter_Parameters_Belt.BRDResistorValue := 1000; // = 100,0 ohm, this is the minimum value
SettingsT02W06.Inverter_Parameters_Belt.FreeRunStop := FALSE;
SettingsT02W06.Inverter_Parameters_Belt.UsageRateOfRegenerativeBraking := 0;
SettingsT02W06.Inverter_Parameters_Belt.UseExternalBrakeResistor := FALSE;

SettingsT02W06.Inverter_NodeNumber_Track := 24;
SettingsT02W06.Inverter_Parameters_Track.AccelerationTime := 100;
SettingsT02W06.Inverter_Parameters_Track.DecelerationTime := 100;
SettingsT02W06.Inverter_Parameters_Track.MAXFrequency := 870;
SettingsT02W06.Inverter_Parameters_Track.MotorCapacity := 2;
SettingsT02W06.Inverter_Parameters_Track.MotorCurrent := 506;
SettingsT02W06.Inverter_Parameters_Track.BrakeONFrequency := 0;
SettingsT02W06.Inverter_Parameters_Track.BrakeReleaseCurrent := 0;
SettingsT02W06.Inverter_Parameters_Track.BrakeReleaseFrequency := 0;
SettingsT02W06.Inverter_Parameters_Track.BRDResistorValue := 1000; // = 100,0 ohm, this is the minimum value
SettingsT02W06.Inverter_Parameters_Track.FreeRunStop := FALSE;
SettingsT02W06.Inverter_Parameters_Track.UsageRateOfRegenerativeBraking := 0;
SettingsT02W06.Inverter_Parameters_Track.UseExternalBrakeResistor := FALSE;

SettingsT02W06.ForwardIsInput := FALSE;
SettingsT02W06.MaxSpeed := 3500;
SettingsT02W06.MinSpeed := 1500;
SettingsT02W06.TimeHighSpeed := 100;
SettingsT02W06.MAX_Run_Time := 600;
SettingsT02W06.TimeDelayON_IS201 := 1;
SettingsT02W06.TimeDelayOFF_IS201 := 20;
SettingsT02W06.TimeDelayON_IS202 := 1;
SettingsT02W06.TimeDelayOFF_IS202 := 20;
SettingsT02W06.TimeDelayON_ISPresent := 5;
SettingsT02W06.TimeDelayOFF_ISPresent := 20;
SettingsT02W06.TimeDelayON_LSTrackDown := 20;
SettingsT02W06.TimeDelayON_LSTrackUp := 20;
SettingsT02W06.TrackDirection := T02W06_Direction;
SettingsT02W06.UsePushButton := FALSE;
SettingsT02W06.UseInstructionTrack := FALSE;
SettingsT02W06.MaxSpeedBelt := 5000;
SettingsT02W06.MinSpeedBelt := 3500;
SettingsT02W06.TimeHighSpeedBelt := 120;
SettingsT02W06.HardwareCodeBuffer:= 202;
SettingsT02W06.DoTransferInbound_101:= TRUE;
SettingsT02W06.DoTransferOutbound_101:= TRUE;
SettingsT02W06.DoTransferInbound201_Buffer:= FALSE; // Must be false as soon as BoweryOS and Dat-A-Control 
SettingsT02W06.DoTransferOutbound201_Buffer:= FALSE;
SettingsT02W06.DoTransferInbound202_Buffer := FALSE;
SettingsT02W06.DoTransferOutbound202_Buffer := TRUE;
SettingsT02W06.DoubleSolenoidValve:= TRUE;

